	{attribute 'export' := '("archive":"True","communication":("cycle":"base","unsubscribe":["setpoint.LLV","setpoint.L1V","setpoint.LV","setpoint.HV","setpoint.H1V","setpoint.HHV"]),"journal":"True","name":("full":"Температура воздуха на входе осевого компрессора","short":"t на вх. Д"),"unit":("engineering":"°С","electrical":"°С"),"digit":"1","connection":("module":"UCP1-A1-AI7-5","type":"R","device_clamp":"UCP1","clamp":"XAI6:9A XAI6:9B XAI6:10B"),"subsystem":"Блок двигателя","group":["Блок двигателя"])'}
	Ta_inK : Taipar := (setpoint := (activation_flags := 0, hyst := GVL_LIB.Hyst_SP), cfg := (par_type := 4, lolim := -100, hilim := 200)); //Температура воздуха на входе осевого компрессора///Уставки//
END_VAR
(* global variable list aopar *)
{region INFO}
(*
 Назначение: Используется для хранения, инициализации и передачи на ВУ значений и состояния выходных аналоговых параметров
 Автор:      /Andrey/ 16.07.2025 17:15:05
 Версия ТЭ5: v00.00.01
 Проект:     KA107
*)
{endregion}
{attribute 'qualified_only'}
{attribute 'symbol' := 'readwrite'}
VAR_GLOBAL
	{attribute 'symbol' := 'none'}
	common : Taopar;
	{attribute 'export' := '("archive":"True","communication":("cycle":"fast"),"journal":"True","name":("full":"Управление положением дозатора газа"),"unit":("engineering":"%"),"connection":("module":"UCP1-A2-AO1-1","type":"I, акт.","device_clamp":"UCP1","clamp":"FVPP1:1 FVPP1:2"),"subsystem":"Блок двигателя","group":["Блок двигателя"])'}
	DG_set : Taopar := (cfg := (par_type := 1, lolim := 0, hilim := 100)); //Управление положением дозатора газа//
END_VAR
(* global variable list dipar *)
{region INFO}
(*
 Назначение: Используется для хранения, инициализации и передачи на ВУ значений и состояния входных дискретных параметров
 Автор:      /Andrey/ 16.07.2025 17:15:05
 Версия ТЭ5: v00.00.01
 Проект:     KA107
*)
{endregion}
{attribute 'qualified_only'}
{attribute 'symbol' := 'readwrite'}
VAR_GLOBAL
	{attribute 'symbol' := 'none'}
	common : Tdipar;

	{attribute 'symbol' := 'none'}
	AO_BA_ai : Tai_to_di;
	{attribute 'export' := '("archive":"True","communication":("cycle":"base"),"journal":"True","name":("full":"АО от блока автоматики ГПА"),"connection":("module":"UCP1-A2-DI1-01","type":"НО СК","device_clamp":"UCP1","clamp":"XDI1:1A XDI1:1B"),"subsystem":"Блок автоматики","group":["Блок автоматики"])'}
	AO_BA : Tdipar; //АО от блока автоматики ГПА//

	{attribute 'symbol' := 'none'}
	Fire_OD_ai : Tai_to_di;
	{attribute 'export' := '("archive":"True","communication":("cycle":"base"),"journal":"True","name":("full":"Пожар ОД"),"connection":("module":"UCP1-A2-DI1-02","type":"НО СК","device_clamp":"UCP1","clamp":"XDI1:2A XDI1:2B"),"subsystem":"Блок автоматики","group":["Блок автоматики"])'}
	Fire_OD : Tdipar; //Пожар ОД//

	{attribute 'symbol' := 'none'}
	Lm_MB_Pn_ai : Tai_to_di;
	{attribute 'export' := '("archive":"True","communication":("cycle":"base"),"journal":"True","name":("full":"Уровень масла в МБД+Н минимальный"),"connection":("module":"UCP1-A2-DI1-05","type":"НО СК","device_clamp":"UCP1","clamp":"XDI1:5A XDI1:5B"),"subsystem":"Маслосистема Д","group":["Маслосистема Д"])'}
	Lm_MB_Pn : Tdipar; //Уровень масла в МБД+Н минимальный//

	{attribute 'symbol' := 'none'}
	Lm_MBU_Pn_ai : Tai_to_di;
	{attribute 'export' := '("archive":"True","communication":("cycle":"base"),"journal":"True","name":("full":"Уровень масла в МБУпл. минимальный"),"connection":("module":"UCP1-A2-DI1-06","type":"НО СК","device_clamp":"UCP1","clamp":"XDI1:6A XDI1:6B"),"subsystem":"Маслосистема К","group":["Маслосистема К"])'}
	Lm_MBU_Pn : Tdipar; //Уровень масла в МБУпл. минимальный//

	{attribute 'symbol' := 'none'}
	Zagaz_OD_Pv_ai : Tai_to_di;
	{attribute 'export' := '("archive":"True","communication":("cycle":"base"),"journal":"True","name":("full":"Загазованность контейнеров выше нормы"),"connection":("module":"UCP1-A2-DI1-07","type":"НО СК","device_clamp":"UCP1","clamp":"XDI1:7A XDI1:7B"),"subsystem":"Блок автоматики","group":["Блок автоматики"])'}
	Zagaz_OD_Pv : Tdipar; //Загазованность контейнеров выше нормы//

	{attribute 'symbol' := 'none'}
	SurgeD_ai : Tai_to_di;
	{attribute 'export' := '("archive":"True","communication":("cycle":"base"),"journal":"True","name":("full":"Помпаж двигателя"),"connection":("module":"UCP1-A2-DI1-09","type":"НО СК","device_clamp":"UCP1","clamp":"XDI1:9A XDI1:9B"),"subsystem":"Блок двигателя","group":["Блок двигателя"])'}
	SurgeD : Tdipar; //Помпаж двигателя//

	{attribute 'symbol' := 'none'}
	Pm_TK_An_ai : Tai_to_di;
	{attribute 'export' := '("archive":"True","communication":("cycle":"base"),"journal":"True","name":("full":"Давление масла смазки ТК аварийная"),"connection":("module":"UCP1-A2-DI1-10","type":"НО СК","device_clamp":"UCP1","clamp":"XDI1:10A XDI1:10B"),"subsystem":"Блок двигателя","group":["Блок двигателя"])'}
	Pm_TK_An : Tdipar; //Давление масла смазки ТК аварийная//

	{attribute 'symbol' := 'none'}
	Pm_ST_An_ai : Tai_to_di;
	{attribute 'export' := '("archive":"True","communication":("cycle":"base"),"journal":"True","name":("full":"Давление масла смазки СТ аварийная"),"connection":("module":"UCP1-A2-DI1-11","type":"НО СК","device_clamp":"UCP1","clamp":"XDI1:11A XDI1:11B"),"subsystem":"Блок двигателя","group":["Блок двигателя"])'}
	Pm_ST_An : Tdipar; //Давление масла смазки СТ аварийная//

	{attribute 'symbol' := 'none'}
	Pm_N_An_ai : Tai_to_di;
	{attribute 'export' := '("archive":"True","communication":("cycle":"base"),"journal":"True","name":("full":"Давление масла смазки Н аварийная"),"connection":("module":"UCP1-A2-DI1-12","type":"НО СК","device_clamp":"UCP1","clamp":"XDI1:12A XDI1:12B"),"subsystem":"Блок компрессора","group":["Блок компрессора"])'}
	Pm_N_An : Tdipar; //Давление масла смазки Н аварийная//

	{attribute 'symbol' := 'none'}
	dPmg_An_ai : Tai_to_di;
	{attribute 'export' := '("archive":"True","communication":("cycle":"base"),"journal":"True","name":("full":"Аварийный перепад масло-газ"),"connection":("module":"UCP1-A2-DI1-13","type":"НО СК","device_clamp":"UCP1","clamp":"XDI1:13A XDI1:13B"),"subsystem":"Блок компрессора","group":["Блок компрессора"])'}
	dPmg_An : Tdipar; //Аварийный перепад масло-газ//

	{attribute 'symbol' := 'none'}
	Pm_SAR_An_ai : Tai_to_di;
	{attribute 'export' := '("archive":"True","communication":("cycle":"base"),"journal":"True","name":("full":"Давление масла САР < 1,5 МПа"),"connection":("module":"UCP1-A2-DI1-14","type":"НО СК","device_clamp":"UCP1","clamp":"XDI1:14A XDI1:14B"),"subsystem":"Блок двигателя","group":["Блок двигателя"])'}
	Pm_SAR_An : Tdipar; //Давление масла САР < 1,5 МПа//

	{attribute 'symbol' := 'none'}
	dP_F_Pv_ai : Tai_to_di;
	{attribute 'export' := '("archive":"True","communication":("cycle":"base"),"journal":"True","name":("full":"dP перед форсунками камеры сгорания >10кПа"),"connection":("module":"UCP1-A2-DI2-15","type":"НО СК","device_clamp":"UCP1","clamp":"FVD2:6 FVD2:5"),"subsystem":"Блок двигателя","group":["Блок двигателя"])'}
	dP_F_Pv : Tdipar; //dP перед форсунками камеры сгорания >10кПа//

	{attribute 'export' := '("archive":"True","communication":("cycle":"base"),"journal":"True","name":("full":"Вентилятор АВОМД+Н+У №1 включен"),"connection":("module":"UCP1-A2-DI3-3","type":"НО СК","device_clamp":"UCP1","clamp":"XDI2:3A XDI2:3B"),"subsystem":"АВОМ","group":["АВОМ"])'}
	Vn1_AVOM_ON : Tdipar; //Вентилятор АВОМД+Н+У №1 включен//
	{attribute 'export' := '("archive":"True","communication":("cycle":"base"),"journal":"True","name":("full":"Вентилятор АВОМД+Н+У №2 включен"),"connection":("module":"UCP1-A2-DI3-4","type":"НО СК","device_clamp":"UCP1","clamp":"XDI2:4A XDI2:4B"),"subsystem":"АВОМ","group":["АВОМ"])'}
	Vn2_AVOM_ON : Tdipar; //Вентилятор АВОМД+Н+У №2 включен//
	{attribute 'export' := '("archive":"True","communication":("cycle":"base"),"journal":"True","name":("full":"Вентилятор ВОУ включен"),"connection":("module":"UCP1-A2-DI3-5","type":"НО СК","device_clamp":"UCP1","clamp":"XDI2:5A XDI2:5B"),"subsystem":"Блок автоматики","group":["Блок автоматики"])'}
	VV_VOU_ON : Tdipar; //Вентилятор ВОУ включен//
	{attribute 'export' := '("archive":"True","communication":("cycle":"base"),"journal":"True","name":("full":"Вытяжной вентилятор нагнетателя ВВН включен"),"connection":("module":"UCP1-A2-DI3-6","type":"НО СК","device_clamp":"UCP1","clamp":"XDI2:6A XDI2:6B"),"subsystem":"Блок автоматики","group":["Блок автоматики"])'}
	VVN_ON : Tdipar; //Вытяжной вентилятор нагнетателя ВВН включен//
	{attribute 'export' := '("archive":"True","communication":("cycle":"base"),"journal":"True","name":("full":"ТРК: готовность"),"connection":("module":"UCP1-A2-DI3-9","type":"НО СК","device_clamp":"UCP1","clamp":"XDI2:9A XDI2:9B"),"subsystem":"Блок двигателя","group":["Блок двигателя"])'}
	TRKready : Tdipar; //ТРК: готовность//
	{attribute 'export' := '("archive":"True","communication":("cycle":"base"),"journal":"True","name":("full":"ТРК: авария"),"connection":("module":"UCP1-A2-DI3-10","type":"НЗ СК","device_clamp":"UCP1","clamp":"XDI2:10A XDI2:10B"),"subsystem":"Блок двигателя","group":["Блок двигателя"])'}
	TRKalr : Tdipar := (inv := TRUE); //ТРК: авария//
	{attribute 'export' := '("archive":"True","communication":("cycle":"base"),"journal":"True","name":("full":"Давление газа перед дозатором газа Предупредительное"),"connection":("module":"UCP1-A2-DI3-18","type":"НЗ СК","device_clamp":"UCP1","clamp":"XDI2:18A XDI2:18B"),"subsystem":"Блок двигателя","group":["Блок двигателя"])'}
	Ptg_inDG_Pn : Tdipar := (inv := TRUE); //Давление газа перед дозатором газа Предупредительное//
	{attribute 'export' := '("archive":"True","communication":("cycle":"base"),"journal":"True","name":("full":"Вентилятор АВОМД+Н+У №3 включен"),"connection":("module":"UCP1-A2-DI3-22","type":"НО СК","device_clamp":"UCP1","clamp":"XDI2:22A XDI2:22B"),"subsystem":"АВОМ","group":["АВОМ"])'}
	Vn3_AVOM_ON : Tdipar; //Вентилятор АВОМД+Н+У №3 включен//
	{attribute 'export' := '("archive":"True","communication":("cycle":"base"),"journal":"True","name":("full":"Вентилятор АВОМД+Н+У №4 включен"),"connection":("module":"UCP1-A2-DI3-23","type":"НО СК","device_clamp":"UCP1","clamp":"XDI2:23A XDI2:23B"),"subsystem":"АВОМ","group":["АВОМ"])'}
	Vn4_AVOM_ON : Tdipar; //Вентилятор АВОМД+Н+У №4 включен//
	{attribute 'export' := '("archive":"True","communication":("cycle":"base"),"journal":"True","name":("full":"Давление газа перед дозатором газа Аварийное"),"connection":("module":"UCP1-A2-DI3-24","type":"НО СК","device_clamp":"UCP1","clamp":"XDI2:24A XDI2:24B"),"subsystem":"Блок топливного газа","group":["Блок топливного газа"])'}
	Ptg_inDG_An : Tdipar; //Давление газа перед дозатором газа Аварийное//
	{attribute 'export' := '("archive":"True","communication":("cycle":"base"),"journal":"True","name":("full":"диаг. Предохранитель UCP1-XTFU1:1 питания модулей AO исправен"),"connection":("module":"UCP1-A2-DI4-17","type":"НО СК","device_clamp":"UCP1","clamp":"Внутр. сигнал"),"subsystem":"Блок автоматики","group":["Блок автоматики"])'}
	Fuse_AO_UCP1 : Tdipar; //диаг. Предохранитель UCP1-XTFU1:1 питания модулей AO исправен//
	{attribute 'export' := '("archive":"True","communication":("cycle":"base"),"journal":"True","name":("full":"диаг. Предохранитель UCP1-XTFU1:2 питания модулей DO исправен"),"connection":("module":"UCP1-A2-DI4-18","type":"НО СК","device_clamp":"UCP1","clamp":"Внутр. сигнал"),"subsystem":"Блок автоматики","group":["Блок автоматики"])'}
	Fuse_DO_UCP1 : Tdipar; //диаг. Предохранитель UCP1-XTFU1:2 питания модулей DO исправен//
	{attribute 'export' := '("archive":"True","communication":("cycle":"base"),"journal":"True","name":("full":"диаг. Предохранитель UCP1--XTFU6:1 питания датчиков температуры и влажности"),"connection":("module":"UCP1-A2-DI4-19","type":"НО СК","device_clamp":"UCP1","clamp":"Внутр. сигнал"),"subsystem":"Блок автоматики","group":["Блок автоматики"])'}
	Fuse_Air_UCP1 : Tdipar; //диаг. Предохранитель UCP1--XTFU6:1 питания датчиков температуры и влажности//
	{attribute 'symbol' := 'none'}
	AO_PRU_1_ai : Tai_to_di;
	{attribute 'export' := '("archive":"True","communication":("cycle":"base"),"journal":"True","name":("full":"Кнопка АО на ПРУ сигнал 1 (НР)"),"connection":("module":"UE1-A1-DI1-01","type":"НО СК","device_clamp":"UE1","clamp":"XTH1:4 XTH1:3"),"subsystem":"Блок автоматики","group":["Блок автоматики"])'}
	AO_PRU_1 : Tdipar; //Кнопка АО на ПРУ сигнал 1 (НР)//

	{attribute 'symbol' := 'none'}
	Kr1_off_ai : Tai_to_di;
	{attribute 'export' := '("archive":"True","communication":("cycle":"base"),"journal":"True","name":("full":"Кран 1 закрыт"),"connection":("module":"UE1-A1-DI1-02","type":"НО СК","device_clamp":"UE1","clamp":"XDI1:2A XDI1:2B"),"subsystem":"Газовая обвязка","group":["Газовая обвязка"])'}
	Kr1_off : Tdipar; //Кран 1 закрыт//

	{attribute 'symbol' := 'none'}
	Kr2_off_ai : Tai_to_di;
	{attribute 'export' := '("archive":"True","communication":("cycle":"base"),"journal":"True","name":("full":"Кран 2 закрыт"),"connection":("module":"UE1-A1-DI1-03","type":"НО СК","device_clamp":"UE1","clamp":"XDI1:3A XDI1:3B"),"subsystem":"Газовая обвязка","group":["Газовая обвязка"])'}
	Kr2_off : Tdipar; //Кран 2 закрыт//

	{attribute 'symbol' := 'none'}
	Kr4_off_ai : Tai_to_di;
	{attribute 'export' := '("archive":"True","communication":("cycle":"base"),"journal":"True","name":("full":"Кран 4 закрыт"),"connection":("module":"UE1-A1-DI1-04","type":"НО СК","device_clamp":"UE1","clamp":"XDI1:4A XDI1:4B"),"subsystem":"Газовая обвязка","group":["Газовая обвязка"])'}
	Kr4_off : Tdipar; //Кран 4 закрыт//

	{attribute 'symbol' := 'none'}
	Kr5_off_ai : Tai_to_di;
	{attribute 'export' := '("archive":"True","communication":("cycle":"base"),"journal":"True","name":("full":"Кран 5 закрыт"),"connection":("module":"UE1-A1-DI1-05","type":"НО СК","device_clamp":"UE1","clamp":"XDI1:5A XDI1:5B"),"subsystem":"Газовая обвязка","group":["Газовая обвязка"])'}
	Kr5_off : Tdipar; //Кран 5 закрыт//

	{attribute 'symbol' := 'none'}
	Kr6_off_ai : Tai_to_di;
	{attribute 'export' := '("archive":"True","communication":("cycle":"base"),"journal":"True","name":("full":"Кран 6 закрыт"),"connection":("module":"UE1-A1-DI1-06","type":"НО СК","device_clamp":"UE1","clamp":"XDI1:6A XDI1:6B"),"subsystem":"Газовая обвязка","group":["Газовая обвязка"])'}
	Kr6_off : Tdipar; //Кран 6 закрыт//

	{attribute 'symbol' := 'none'}
	Kr12_off_ai : Tai_to_di;
	{attribute 'export' := '("archive":"True","communication":("cycle":"base"),"journal":"True","name":("full":"Кран 12 закрыт (т.г.)"),"connection":("module":"UE1-A1-DI1-07","type":"НО СК","device_clamp":"UE1","clamp":"XDI1:7A XDI1:7B"),"subsystem":"Газовая обвязка","group":["Газовая обвязка"])'}
	Kr12_off : Tdipar; //Кран 12 закрыт (т.г.)//

	{attribute 'symbol' := 'none'}
	Kr9_off_ai : Tai_to_di;
	{attribute 'export' := '("archive":"True","communication":("cycle":"base"),"journal":"True","name":("full":"Кран 9 закрыт (т.газ. свеча.)"),"connection":("module":"UE1-A1-DI1-08","type":"НО СК","device_clamp":"UE1","clamp":"XDI1:8A XDI1:8B"),"subsystem":"Газовая обвязка","group":["Газовая обвязка"])'}
	Kr9_off : Tdipar; //Кран 9 закрыт (т.газ. свеча.)//

	{attribute 'symbol' := 'none'}
	Kr11_off_ai : Tai_to_di;
	{attribute 'export' := '("archive":"True","communication":("cycle":"base"),"journal":"True","name":("full":"Кран 11 закрыт (п.г.)"),"connection":("module":"UE1-A1-DI1-09","type":"НО СК","device_clamp":"UE1","clamp":"XDI1:9A XDI1:9B"),"subsystem":"Газовая обвязка","group":["Газовая обвязка"])'}
	Kr11_off : Tdipar; //Кран 11 закрыт (п.г.)//

	{attribute 'symbol' := 'none'}
	Kr10_off_ai : Tai_to_di;
	{attribute 'export' := '("archive":"True","communication":("cycle":"base"),"journal":"True","name":("full":"Кран 10 закрыт (п.газ. свеча.)"),"connection":("module":"UE1-A1-DI1-10","type":"НО СК","device_clamp":"UE1","clamp":"XDI1:10A XDI1:10B"),"subsystem":"Газовая обвязка","group":["Газовая обвязка"])'}
	Kr10_off : Tdipar; //Кран 10 закрыт (п.газ. свеча.)//

	{attribute 'symbol' := 'none'}
	KPV1_off_ai : Tai_to_di;
	{attribute 'export' := '("archive":"True","communication":("cycle":"base"),"journal":"True","name":("full":"КПВ-1 закрыт"),"connection":("module":"UE1-A1-DI1-11","type":"НО СК","device_clamp":"UE1","clamp":"XDI1:11A XDI1:11B"),"subsystem":"Блок двигателя","group":["Блок двигателя"])'}
	KPV1_off : Tdipar; //КПВ-1 закрыт//

	{attribute 'symbol' := 'none'}
	KPV2_off_ai : Tai_to_di;
	{attribute 'export' := '("archive":"True","communication":("cycle":"base"),"journal":"True","name":("full":"КПВ-2 закрыт"),"connection":("module":"UE1-A1-DI1-12","type":"НО СК","device_clamp":"UE1","clamp":"XDI1:12A XDI1:12B"),"subsystem":"Блок двигателя","group":["Блок двигателя"])'}
	KPV2_off : Tdipar; //КПВ-2 закрыт//

	{attribute 'symbol' := 'none'}
	KPV3_off_ai : Tai_to_di;
	{attribute 'export' := '("archive":"True","communication":("cycle":"base"),"journal":"True","name":("full":"КПВ-3 закрыт"),"connection":("module":"UE1-A1-DI1-13","type":"НО СК","device_clamp":"UE1","clamp":"XDI1:13A XDI1:13B"),"subsystem":"Блок двигателя","group":["Блок двигателя"])'}
	KPV3_off : Tdipar; //КПВ-3 закрыт//

	{attribute 'symbol' := 'none'}
	KPV4_off_ai : Tai_to_di;
	{attribute 'export' := '("archive":"True","communication":("cycle":"base"),"journal":"True","name":("full":"КПВ-4 закрыт"),"connection":("module":"UE1-A1-DI1-14","type":"НО СК","device_clamp":"UE1","clamp":"XDI1:14A XDI1:14B"),"subsystem":"Блок двигателя","group":["Блок двигателя"])'}
	KPV4_off : Tdipar; //КПВ-4 закрыт//

	{attribute 'symbol' := 'none'}
	KPV5_off_ai : Tai_to_di;
	{attribute 'export' := '("archive":"True","communication":("cycle":"base"),"journal":"True","name":("full":"КПВ-5 закрыт"),"connection":("module":"UE1-A1-DI1-15","type":"НО СК","device_clamp":"UE1","clamp":"XDI1:15A XDI1:15B"),"subsystem":"Блок двигателя","group":["Блок двигателя"])'}
	KPV5_off : Tdipar; //КПВ-5 закрыт//

	{attribute 'symbol' := 'none'}
	SK_off_ai : Tai_to_di;
	{attribute 'export' := '("archive":"True","communication":("cycle":"fast"),"journal":"True","name":("full":"СК закрыт"),"connection":("module":"UE1-A1-DI1-16","type":"НО СК","device_clamp":"UE1","clamp":"XDI1:16A XDI1:16B"),"subsystem":"Блок топливного газа","group":["Блок топливного газа"])'}
	SK_off : Tdipar; //СК закрыт//

	{attribute 'symbol' := 'none'}
	AO_PRU_2_ai : Tai_to_di;
	{attribute 'export' := '("archive":"True","communication":("cycle":"base"),"journal":"True","name":("full":"Кнопка АО на ПРУ сигнал 2 (НЗ)"),"connection":("module":"UE1-A1-DI2-01","type":"НЗ СК","device_clamp":"UE1","clamp":"XTH1:13 XTH1:14"),"subsystem":"Блок автоматики","group":["Блок автоматики"])'}
	AO_PRU_2 : Tdipar := (inv := TRUE); //Кнопка АО на ПРУ сигнал 2 (НЗ)//

	{attribute 'symbol' := 'none'}
	Kr1_ON_ai : Tai_to_di;
	{attribute 'export' := '("archive":"True","communication":("cycle":"base"),"journal":"True","name":("full":"Кран 1 открыт"),"connection":("module":"UE1-A1-DI2-02","type":"НО СК","device_clamp":"UE1","clamp":"XDI1:18A XDI1:18B"),"subsystem":"Газовая обвязка","group":["Газовая обвязка"])'}
	Kr1_ON : Tdipar; //Кран 1 открыт//

	{attribute 'symbol' := 'none'}
	Kr2_ON_ai : Tai_to_di;
	{attribute 'export' := '("archive":"True","communication":("cycle":"base"),"journal":"True","name":("full":"Кран 2 открыт"),"connection":("module":"UE1-A1-DI2-03","type":"НО СК","device_clamp":"UE1","clamp":"XDI1:19A XDI1:19B"),"subsystem":"Газовая обвязка","group":["Газовая обвязка"])'}
	Kr2_ON : Tdipar; //Кран 2 открыт//

	{attribute 'symbol' := 'none'}
	Kr4_ON_ai : Tai_to_di;
	{attribute 'export' := '("archive":"True","communication":("cycle":"base"),"journal":"True","name":("full":"Кран 4 открыт"),"connection":("module":"UE1-A1-DI2-04","type":"НО СК","device_clamp":"UE1","clamp":"XDI1:20A XDI1:20B"),"subsystem":"Газовая обвязка","group":["Газовая обвязка"])'}
	Kr4_ON : Tdipar; //Кран 4 открыт//

	{attribute 'symbol' := 'none'}
	Kr5_ON_ai : Tai_to_di;
	{attribute 'export' := '("archive":"True","communication":("cycle":"base"),"journal":"True","name":("full":"Кран 5 открыт"),"connection":("module":"UE1-A1-DI2-05","type":"НО СК","device_clamp":"UE1","clamp":"XDI1:21A XDI1:21B"),"subsystem":"Газовая обвязка","group":["Газовая обвязка"])'}
	Kr5_ON : Tdipar; //Кран 5 открыт//

	{attribute 'symbol' := 'none'}
	Kr6_ON_ai : Tai_to_di;
	{attribute 'export' := '("archive":"True","communication":("cycle":"base"),"journal":"True","name":("full":"Кран 6 открыт"),"connection":("module":"UE1-A1-DI2-06","type":"НО СК","device_clamp":"UE1","clamp":"XDI1:22A XDI1:22B"),"subsystem":"Газовая обвязка","group":["Газовая обвязка"])'}
	Kr6_ON : Tdipar; //Кран 6 открыт//

	{attribute 'symbol' := 'none'}
	Kr12_ON_ai : Tai_to_di;
	{attribute 'export' := '("archive":"True","communication":("cycle":"base"),"journal":"True","name":("full":"Кран 12 открыт (т.г.)"),"connection":("module":"UE1-A1-DI2-07","type":"НО СК","device_clamp":"UE1","clamp":"XDI1:23A XDI1:23B"),"subsystem":"Газовая обвязка","group":["Газовая обвязка"])'}
	Kr12_ON : Tdipar; //Кран 12 открыт (т.г.)//

	{attribute 'symbol' := 'none'}
	Kr9_ON_ai : Tai_to_di;
	{attribute 'export' := '("archive":"True","communication":("cycle":"base"),"journal":"True","name":("full":"Кран 9 открыт (т.газ. свеча.)"),"connection":("module":"UE1-A1-DI2-08","type":"НО СК","device_clamp":"UE1","clamp":"XDI1:24A XDI1:24B"),"subsystem":"Газовая обвязка","group":["Газовая обвязка"])'}
	Kr9_ON : Tdipar; //Кран 9 открыт (т.газ. свеча.)//

	{attribute 'symbol' := 'none'}
	Kr11_ON_ai : Tai_to_di;
	{attribute 'export' := '("archive":"True","communication":("cycle":"base"),"journal":"True","name":("full":"Кран 11 открыт (п.г.)"),"connection":("module":"UE1-A1-DI2-09","type":"НО СК","device_clamp":"UE1","clamp":"XDI1:25A XDI1:25B"),"subsystem":"Газовая обвязка","group":["Газовая обвязка"])'}
	Kr11_ON : Tdipar; //Кран 11 открыт (п.г.)//

	{attribute 'symbol' := 'none'}
	Kr10_ON_ai : Tai_to_di;
	{attribute 'export' := '("archive":"True","communication":("cycle":"base"),"journal":"True","name":("full":"Кран 10 открыт (п.газ. свеча.)"),"connection":("module":"UE1-A1-DI2-10","type":"НО СК","device_clamp":"UE1","clamp":"XDI1:26A XDI1:26B"),"subsystem":"Газовая обвязка","group":["Газовая обвязка"])'}
	Kr10_ON : Tdipar; //Кран 10 открыт (п.газ. свеча.)//

	{attribute 'symbol' := 'none'}
	KPV1_ON_ai : Tai_to_di;
	{attribute 'export' := '("archive":"True","communication":("cycle":"base"),"journal":"True","name":("full":"КПВ-1 открыт"),"connection":("module":"UE1-A1-DI2-11","type":"НО СК","device_clamp":"UE1","clamp":"XDI1:27A XDI1:27B"),"subsystem":"Блок двигателя","group":["Блок двигателя"])'}
	KPV1_ON : Tdipar; //КПВ-1 открыт//

	{attribute 'symbol' := 'none'}
	KPV2_ON_ai : Tai_to_di;
	{attribute 'export' := '("archive":"True","communication":("cycle":"base"),"journal":"True","name":("full":"КПВ-2 открыт"),"connection":("module":"UE1-A1-DI2-12","type":"НО СК","device_clamp":"UE1","clamp":"XDI1:28A XDI1:28B"),"subsystem":"Блок двигателя","group":["Блок двигателя"])'}
	KPV2_ON : Tdipar; //КПВ-2 открыт//

	{attribute 'symbol' := 'none'}
	KPV3_ON_ai : Tai_to_di;
	{attribute 'export' := '("archive":"True","communication":("cycle":"base"),"journal":"True","name":("full":"КПВ-3 открыт"),"connection":("module":"UE1-A1-DI2-13","type":"НО СК","device_clamp":"UE1","clamp":"XDI1:29A XDI1:29B"),"subsystem":"Блок двигателя","group":["Блок двигателя"])'}
	KPV3_ON : Tdipar; //КПВ-3 открыт//

	{attribute 'symbol' := 'none'}
	KPV4_ON_ai : Tai_to_di;
	{attribute 'export' := '("archive":"True","communication":("cycle":"base"),"journal":"True","name":("full":"КПВ-4 открыт"),"connection":("module":"UE1-A1-DI2-14","type":"НО СК","device_clamp":"UE1","clamp":"XDI1:30A XDI1:30B"),"subsystem":"Блок двигателя","group":["Блок двигателя"])'}
	KPV4_ON : Tdipar; //КПВ-4 открыт//

	{attribute 'symbol' := 'none'}
	KPV5_ON_ai : Tai_to_di;
	{attribute 'export' := '("archive":"True","communication":("cycle":"base"),"journal":"True","name":("full":"КПВ-5 открыт"),"connection":("module":"UE1-A1-DI2-15","type":"НО СК","device_clamp":"UE1","clamp":"XDI1:31A XDI1:31B"),"subsystem":"Блок двигателя","group":["Блок двигателя"])'}
	KPV5_ON : Tdipar; //КПВ-5 открыт//

	{attribute 'symbol' := 'none'}
	SK_ON_ai : Tai_to_di;
	{attribute 'export' := '("archive":"True","communication":("cycle":"fast"),"journal":"True","name":("full":"СК открыт"),"connection":("module":"UE1-A1-DI2-16","type":"НО СК","device_clamp":"UE1","clamp":"XDI1:32A XDI1:32B"),"subsystem":"Блок топливного газа","group":["Блок топливного газа"])'}
	SK_ON : Tdipar; //СК открыт//

	{attribute 'symbol' := 'none'}
	PNS_ON_ai : Tai_to_di;
	{attribute 'export' := '("archive":"True","communication":("cycle":"base"),"journal":"True","name":("full":"Пусковой насос смазки включен"),"connection":("module":"UE1-A1-DI3-01","type":"НО СК","device_clamp":"UE1","clamp":"XDI2:1A XDI2:1B"),"subsystem":"Маслосистема Д","group":["Маслосистема Д"])'}
	PNS_ON : Tdipar; //Пусковой насос смазки включен//

	{attribute 'symbol' := 'none'}
	PNU_ON_ai : Tai_to_di;
	{attribute 'export' := '("archive":"True","communication":("cycle":"base"),"journal":"True","name":("full":"Пусковой насос уплотнения включен"),"connection":("module":"UE1-A1-DI3-02","type":"НО СК","device_clamp":"UE1","clamp":"XDI2:2A XDI2:2B"),"subsystem":"Маслосистема К","group":["Маслосистема К"])'}
	PNU_ON : Tdipar; //Пусковой насос уплотнения включен//

	{attribute 'export' := '("archive":"True","communication":("cycle":"base"),"journal":"True","name":("full":"Повышенная вибрация двигателя"),"connection":("module":"UE1-A1-DI4-9","type":"НО СК","device_clamp":"UE1","clamp":"XDI3:9A XDI3:9B"),"subsystem":"Блок двигателя","group":["Блок двигателя"])'}
	Vs_D_Pv : Tdipar; //Повышенная вибрация двигателя//
	{attribute 'export' := '("archive":"True","communication":("cycle":"base"),"journal":"True","name":("full":"Опасная вибрация двигателя"),"connection":("module":"UE1-A1-DI4-10","type":"НО СК","device_clamp":"UE1","clamp":"XDI3:10A XDI3:10B"),"subsystem":"Блок двигателя","group":["Блок двигателя"])'}
	Vs_D_Av : Tdipar; //Опасная вибрация двигателя//
	{attribute 'export' := '("archive":"True","communication":("cycle":"base"),"journal":"True","name":("full":"Осевой сдвиг ротора Н Аварийный"),"connection":("module":"UE1-A1-DI4-18","type":"НО СК","device_clamp":"UE1","clamp":"XDI3:18A XDI3:18B"),"subsystem":"Блок компрессора","group":["Блок компрессора"])'}
	Zs_Nl : Tdipar; //Осевой сдвиг ротора Н Аварийный//
	{attribute 'export' := '("archive":"True","communication":("cycle":"base"),"journal":"True","name":("full":"Давление газа после крана 1"),"connection":("module":"UE1-A1-DI4-20","type":"НО СК","device_clamp":"UE1","clamp":"XDI3:20A XDI3:20B"),"subsystem":"Газовая обвязка","group":["Газовая обвязка"])'}
	Pg_outKR1 : Tdipar; //Давление газа после крана 1//
	{attribute 'export' := '("archive":"True","communication":("cycle":"base"),"journal":"True","name":("full":"Давление масла смазки Н предупредительная"),"connection":("module":"UE1-A1-DI4-23","type":"НО СК","device_clamp":"UE1","clamp":"XDI3:23A XDI3:23B"),"subsystem":"Маслосистема К","group":["Маслосистема К"])'}
	Pm_N_Pn : Tdipar; //Давление масла смазки Н предупредительная//
	{attribute 'export' := '("archive":"True","communication":("cycle":"base"),"journal":"True","name":("full":"Разрежение в ВОУ"),"connection":("module":"UE1-A1-DI4-24","type":"НО СК","device_clamp":"UE1","clamp":"XDI3:24A XDI3:24B"),"subsystem":"Блок двигателя","group":["Блок двигателя"])'}
	Exh_VOU : Tdipar; //Разрежение в ВОУ//
	{attribute 'export' := '("archive":"True","communication":("cycle":"base"),"journal":"True","name":("full":"Давление газа до крана 13 (воздушного стартера)"),"connection":("module":"UE1-A1-DI4-25","type":"НО СК","device_clamp":"UE1","clamp":"XDI3:25A XDI3:25B"),"subsystem":"Газовая обвязка","group":["Газовая обвязка"])'}
	Pg_InKR13 : Tdipar; //Давление газа до крана 13 (воздушного стартера)//
	{attribute 'export' := '("archive":"True","communication":("cycle":"base"),"journal":"True","name":("full":"Давление масла смазки воздушного стартера высокий уровень"),"connection":("module":"UE1-A1-DI4-26","type":"НО СК","device_clamp":"UE1","clamp":"XDI3:26A XDI3:26B"),"subsystem":"Маслосистема Д","group":["Маслосистема Д"])'}
	Pm_Starter_Av : Tdipar; //Давление масла смазки воздушного стартера высокий уровень//
	{attribute 'export' := '("archive":"True","communication":("cycle":"base"),"journal":"True","name":("full":"Давление масла смазки воздушного стартера низкий уровень"),"connection":("module":"UE1-A1-DI4-27","type":"НО СК","device_clamp":"UE1","clamp":"XDI3:27A XDI3:27B"),"subsystem":"Маслосистема Д","group":["Маслосистема Д"])'}
	Pm_Starter_An : Tdipar; //Давление масла смазки воздушного стартера низкий уровень//
	{attribute 'export' := '("archive":"True","communication":("cycle":"base"),"journal":"True","name":("full":"Кнопка ЭАО на ПРУ нажата сигнал 1 (НР)"),"connection":("module":"UE1-A1-DI4-29","type":"НО СК","device_clamp":"UE1","clamp":"Внутр. сигнал"),"subsystem":"Блок автоматики","group":["Блок автоматики"])'}
	EAO_PRU_1 : Tdipar; //Кнопка ЭАО на ПРУ нажата сигнал 1 (НР)//
	{attribute 'export' := '("archive":"True","communication":("cycle":"base"),"journal":"True","name":("full":"Кнопка ЭАО на ПРУ нажата сигнал 2 (НЗ)"),"connection":("module":"UE1-A1-DI4-30","type":"НЗ СК","device_clamp":"UE1","clamp":"Внутр. сигнал"),"subsystem":"Блок автоматики","group":["Блок автоматики"])'}
	EAO_PRU_2 : Tdipar := (inv := TRUE); //Кнопка ЭАО на ПРУ нажата сигнал 2 (НЗ)//
	{attribute 'export' := '("archive":"True","communication":("cycle":"base"),"journal":"True","name":("full":"Кнопка ЭАО на ПРУ нажата сигнал 3 (НЗ)"),"connection":("module":"UE1-A1-DI4-31","type":"НЗ СК","device_clamp":"UE1","clamp":"Внутр. сигнал"),"subsystem":"Блок автоматики","group":["Блок автоматики"])'}
	EAO_PRU_3 : Tdipar := (inv := TRUE); //Кнопка ЭАО на ПРУ нажата сигнал 3 (НЗ)//
	{attribute 'export' := '("archive":"True","communication":("cycle":"base"),"journal":"True","name":("full":"БЭАО сработал"),"connection":("module":"UE1-A1-DI4-32","type":"НО СК","device_clamp":"UE1","clamp":"Внутр. сигнал"),"subsystem":"Блок автоматики","group":["Блок автоматики"])'}
	BEAO : Tdipar; //БЭАО сработал//
	{attribute 'export' := '("archive":"True","communication":("cycle":"base"),"journal":"True","name":("full":"Заслонка ВC (кран 13) открыта"),"connection":("module":"UE1-A1-DI5-1","type":"U","device_clamp":"UE1","clamp":"DA1:A2"),"subsystem":"Газовая обвязка","group":["Газовая обвязка"])'}
	Kr13_ON : Tdipar; //Заслонка ВC (кран 13) открыта//
	{attribute 'export' := '("archive":"True","communication":("cycle":"base"),"journal":"True","name":("full":"БЗА. Авария"),"connection":("module":"UE1-A1-DI5-2","type":"НО СК","device_clamp":"UE1","clamp":"Внутр. сигнал"),"subsystem":"Блок автоматики","group":["Блок автоматики"])'}
	BZA_alr : Tdipar; //БЗА. Авария//
	{attribute 'export' := '("archive":"True","communication":("cycle":"base"),"journal":"True","name":("full":"БЗА. Готовность 1"),"connection":("module":"UE1-A1-DI5-3","type":"НО СК","device_clamp":"UE1","clamp":"Внутр. сигнал"),"subsystem":"Блок автоматики","group":["Блок автоматики"])'}
	BZA_ready_1 : Tdipar; //БЗА. Готовность 1//
	{attribute 'export' := '("archive":"True","communication":("cycle":"base"),"journal":"True","name":("full":"БЗА. Готовность 2"),"connection":("module":"UE1-A1-DI5-4","type":"НО СК","device_clamp":"UE1","clamp":"Внутр. сигнал"),"subsystem":"Блок автоматики","group":["Блок автоматики"])'}
	BZA_ready_2 : Tdipar; //БЗА. Готовность 2//
	{attribute 'export' := '("archive":"True","communication":("cycle":"base"),"journal":"True","name":("full":"Контроль питания СС"),"connection":("module":"UE1-A1-DI5-25","type":"НО СК","device_clamp":"UE1","clamp":"Внутр. сигнал"),"subsystem":"Блок автоматики","group":["Блок автоматики"])'}
	U_CC_cntrl : Tdipar; //Контроль питания СС//
	{attribute 'export' := '("archive":"True","communication":("cycle":"base"),"journal":"True","name":("full":"Стружка в масле на выходе Д"),"connection":("module":"UE1-A1-DI5-26","type":"НО СК","device_clamp":"UE1","clamp":"XDI4:26A XDI4:26B"),"subsystem":"Маслосистема Д","group":["Маслосистема Д"])'}
	Chip_outD : Tdipar; //Стружка в масле на выходе Д//
	{attribute 'export' := '("archive":"True","communication":("cycle":"base"),"journal":"True","name":("full":"Сигнализатор обледенения"),"connection":("module":"UE1-A1-DI5-27","type":"НО СК","device_clamp":"UE1","clamp":"XDI4:27A XDI4:27B"),"subsystem":"Блок автоматики","group":["Блок автоматики"])'}
	Ace_alr : Tdipar; //Сигнализатор обледенения//
	{attribute 'export' := '("archive":"True","communication":("cycle":"base"),"journal":"True","name":("full":"диаг. Кран 1 закрыть"),"connection":("module":"UE1-A1-DI6-1","type":"НО СК","device_clamp":"UE1","clamp":"Внутр. сигнал"),"subsystem":"Газовая обвязка","group":["Газовая обвязка"])'}
	kcdo_Kr1_off : Tdipar; //диаг. Кран 1 закрыть//
	{attribute 'export' := '("archive":"True","communication":("cycle":"base"),"journal":"True","name":("full":"диаг. Кран 1 смазка"),"connection":("module":"UE1-A1-DI6-2","type":"НО СК","device_clamp":"UE1","clamp":"Внутр. сигнал"),"subsystem":"Газовая обвязка","group":["Газовая обвязка"])'}
	kcdo_Kr1m_ON : Tdipar; //диаг. Кран 1 смазка//
	{attribute 'export' := '("archive":"True","communication":("cycle":"base"),"journal":"True","name":("full":"диаг. Кран 2 закрыть"),"connection":("module":"UE1-A1-DI6-3","type":"НО СК","device_clamp":"UE1","clamp":"Внутр. сигнал"),"subsystem":"Газовая обвязка","group":["Газовая обвязка"])'}
	kcdo_Kr2_off : Tdipar; //диаг. Кран 2 закрыть//
	{attribute 'export' := '("archive":"True","communication":("cycle":"base"),"journal":"True","name":("full":"диаг. Кран 2 смазка"),"connection":("module":"UE1-A1-DI6-4","type":"НО СК","device_clamp":"UE1","clamp":"Внутр. сигнал"),"subsystem":"Газовая обвязка","group":["Газовая обвязка"])'}
	kcdo_Kr2m_ON : Tdipar; //диаг. Кран 2 смазка//
	{attribute 'export' := '("archive":"True","communication":("cycle":"base"),"journal":"True","name":("full":"диаг. Кран 4 закрыть"),"connection":("module":"UE1-A1-DI6-5","type":"НО СК","device_clamp":"UE1","clamp":"Внутр. сигнал"),"subsystem":"Газовая обвязка","group":["Газовая обвязка"])'}
	kcdo_Kr4_off : Tdipar; //диаг. Кран 4 закрыть//
	{attribute 'export' := '("archive":"True","communication":("cycle":"base"),"journal":"True","name":("full":"диаг. Кран 4 смазка"),"connection":("module":"UE1-A1-DI6-6","type":"НО СК","device_clamp":"UE1","clamp":"Внутр. сигнал"),"subsystem":"Газовая обвязка","group":["Газовая обвязка"])'}
	kcdo_Kr4m_ON : Tdipar; //диаг. Кран 4 смазка//
	{attribute 'export' := '("archive":"True","communication":("cycle":"base"),"journal":"True","name":("full":"диаг. Кран 5 открыть"),"connection":("module":"UE1-A1-DI6-7","type":"НО СК","device_clamp":"UE1","clamp":"Внутр. сигнал"),"subsystem":"Газовая обвязка","group":["Газовая обвязка"])'}
	kcdo_Kr5_ON : Tdipar; //диаг. Кран 5 открыть//
	{attribute 'export' := '("archive":"True","communication":("cycle":"base"),"journal":"True","name":("full":"диаг. Кран 5 смазка"),"connection":("module":"UE1-A1-DI6-8","type":"НО СК","device_clamp":"UE1","clamp":"Внутр. сигнал"),"subsystem":"Газовая обвязка","group":["Газовая обвязка"])'}
	kcdo_Kr5m_ON : Tdipar; //диаг. Кран 5 смазка//
	{attribute 'export' := '("archive":"True","communication":("cycle":"base"),"journal":"True","name":("full":"диаг. Кран 6 закрыть"),"connection":("module":"UE1-A1-DI6-9","type":"НО СК","device_clamp":"UE1","clamp":"Внутр. сигнал"),"subsystem":"Газовая обвязка","group":["Газовая обвязка"])'}
	kcdo_Kr6_off : Tdipar; //диаг. Кран 6 закрыть//
	{attribute 'export' := '("archive":"True","communication":("cycle":"base"),"journal":"True","name":("full":"диаг. Кран 6 смазка"),"connection":("module":"UE1-A1-DI6-10","type":"НО СК","device_clamp":"UE1","clamp":"Внутр. сигнал"),"subsystem":"Газовая обвязка","group":["Газовая обвязка"])'}
	kcdo_Kr6m_ON : Tdipar; //диаг. Кран 6 смазка//
	{attribute 'export' := '("archive":"True","communication":("cycle":"base"),"journal":"True","name":("full":"диаг. Кран 12 закрыть (т.г.)"),"connection":("module":"UE1-A1-DI6-11","type":"НО СК","device_clamp":"UE1","clamp":"Внутр. сигнал"),"subsystem":"Газовая обвязка","group":["Газовая обвязка"])'}
	kcdo_KR12_off : Tdipar; //диаг. Кран 12 закрыть (т.г.)//
	{attribute 'export' := '("archive":"True","communication":("cycle":"base"),"journal":"True","name":("full":"диаг. Кран 12 смазка"),"connection":("module":"UE1-A1-DI6-12","type":"НО СК","device_clamp":"UE1","clamp":"Внутр. сигнал"),"subsystem":"Газовая обвязка","group":["Газовая обвязка"])'}
	kcdo_KR12m_ON : Tdipar; //диаг. Кран 12 смазка//
	{attribute 'export' := '("archive":"True","communication":("cycle":"base"),"journal":"True","name":("full":"диаг. Кран 9 смазка"),"connection":("module":"UE1-A1-DI6-14","type":"НО СК","device_clamp":"UE1","clamp":"Внутр. сигнал"),"subsystem":"Газовая обвязка","group":["Газовая обвязка"])'}
	kcdo_KR9m_ON : Tdipar; //диаг. Кран 9 смазка//
	{attribute 'export' := '("archive":"True","communication":("cycle":"base"),"journal":"True","name":("full":"диаг. Кран 11 открыть (п.г.)"),"connection":("module":"UE1-A1-DI6-15","type":"НО СК","device_clamp":"UE1","clamp":"Внутр. сигнал"),"subsystem":"Газовая обвязка","group":["Газовая обвязка"])'}
	kcdo_Kr11_ON : Tdipar; //диаг. Кран 11 открыть (п.г.)//
	{attribute 'export' := '("archive":"True","communication":("cycle":"base"),"journal":"True","name":("full":"диаг. Кран 11 смазка"),"connection":("module":"UE1-A1-DI6-16","type":"НО СК","device_clamp":"UE1","clamp":"Внутр. сигнал"),"subsystem":"Газовая обвязка","group":["Газовая обвязка"])'}
	kcdo_Kr11m_ON : Tdipar; //диаг. Кран 11 смазка//
	{attribute 'export' := '("archive":"True","communication":("cycle":"base"),"journal":"True","name":("full":"диаг. Кран 10 смазка"),"connection":("module":"UE1-A1-DI6-18","type":"НО СК","device_clamp":"UE1","clamp":"Внутр. сигнал"),"subsystem":"Газовая обвязка","group":["Газовая обвязка"])'}
	kcdo_Kr10m_ON : Tdipar; //диаг. Кран 10 смазка//
	{attribute 'export' := '("archive":"True","communication":("cycle":"base"),"journal":"True","name":("full":"диаг. Включение КПВ 1,5"),"connection":("module":"UE1-A1-DI6-19","type":"НО СК","device_clamp":"UE1","clamp":"Внутр. сигнал"),"subsystem":"Блок двигателя","group":["Блок двигателя"])'}
	kcdo_KPV15_ON : Tdipar; //диаг. Включение КПВ 1,5//
	{attribute 'export' := '("archive":"True","communication":("cycle":"base"),"journal":"True","name":("full":"диаг. Включение КПВ 2,3"),"connection":("module":"UE1-A1-DI6-20","type":"НО СК","device_clamp":"UE1","clamp":"Внутр. сигнал"),"subsystem":"Блок двигателя","group":["Блок двигателя"])'}
	kcdo_KPV23_off : Tdipar; //диаг. Включение КПВ 2,3//
	{attribute 'export' := '("archive":"True","communication":("cycle":"base"),"journal":"True","name":("full":"диаг. Включение КПВ 4"),"connection":("module":"UE1-A1-DI6-21","type":"НО СК","device_clamp":"UE1","clamp":"Внутр. сигнал"),"subsystem":"Блок двигателя","group":["Блок двигателя"])'}
	kcdo_KPV4_off : Tdipar; //диаг. Включение КПВ 4//
	{attribute 'export' := '("archive":"True","communication":("cycle":"base"),"journal":"True","name":("full":"диаг. Стопорный клапан открыть"),"connection":("module":"UE1-A1-DI6-22","type":"НО СК","device_clamp":"UE1","clamp":"Внутр. сигнал"),"subsystem":"Блок двигателя","group":["Блок двигателя"])'}
	kcdo_SK_ON : Tdipar; //диаг. Стопорный клапан открыть//
	{attribute 'export' := '("archive":"True","communication":("cycle":"base"),"journal":"True","name":("full":"диаг. Кран 1 открыть"),"connection":("module":"UE1-A1-DI7-1","type":"НО СК","device_clamp":"UE1","clamp":"Внутр. сигнал"),"subsystem":"Газовая обвязка","group":["Газовая обвязка"])'}
	kcdo_Kr1_ON : Tdipar; //диаг. Кран 1 открыть//
	{attribute 'export' := '("archive":"True","communication":("cycle":"base"),"journal":"True","name":("full":"диаг. Кран 2 открыть"),"connection":("module":"UE1-A1-DI7-2","type":"НО СК","device_clamp":"UE1","clamp":"Внутр. сигнал"),"subsystem":"Газовая обвязка","group":["Газовая обвязка"])'}
	kcdo_Kr2_ON : Tdipar; //диаг. Кран 2 открыть//
	{attribute 'export' := '("archive":"True","communication":("cycle":"base"),"journal":"True","name":("full":"диаг. Кран 4 открыть"),"connection":("module":"UE1-A1-DI7-3","type":"НО СК","device_clamp":"UE1","clamp":"Внутр. сигнал"),"subsystem":"Газовая обвязка","group":["Газовая обвязка"])'}
	kcdo_Kr4_ON : Tdipar; //диаг. Кран 4 открыть//
	{attribute 'export' := '("archive":"True","communication":("cycle":"base"),"journal":"True","name":("full":"диаг. Кран 5 закрыть"),"connection":("module":"UE1-A1-DI7-4","type":"НО СК","device_clamp":"UE1","clamp":"Внутр. сигнал"),"subsystem":"Газовая обвязка","group":["Газовая обвязка"])'}
	kcdo_Kr5_off : Tdipar; //диаг. Кран 5 закрыть//
	{attribute 'export' := '("archive":"True","communication":("cycle":"base"),"journal":"True","name":("full":"диаг. Кран 6 открыть"),"connection":("module":"UE1-A1-DI7-5","type":"НО СК","device_clamp":"UE1","clamp":"Внутр. сигнал"),"subsystem":"Газовая обвязка","group":["Газовая обвязка"])'}
	kcdo_Kr6_ON : Tdipar; //диаг. Кран 6 открыть//
	{attribute 'export' := '("archive":"True","communication":("cycle":"base"),"journal":"True","name":("full":"диаг. Кран 12 открыть (т.г.)"),"connection":("module":"UE1-A1-DI7-6","type":"НО СК","device_clamp":"UE1","clamp":"Внутр. сигнал"),"subsystem":"Газовая обвязка","group":["Газовая обвязка"])'}
	kcdo_Kr12_ON : Tdipar; //диаг. Кран 12 открыть (т.г.)//
	{attribute 'export' := '("archive":"True","communication":("cycle":"base"),"journal":"True","name":("full":"диаг. Кран 11 закрыть (п.г.)"),"connection":("module":"UE1-A1-DI7-8","type":"НО СК","device_clamp":"UE1","clamp":"Внутр. сигнал"),"subsystem":"Газовая обвязка","group":["Газовая обвязка"])'}
	kcdo_Kr11_off : Tdipar; //диаг. Кран 11 закрыть (п.г.)//
	{attribute 'export' := '("archive":"True","communication":("cycle":"base"),"journal":"True","name":("full":"диаг. ЗВУКОВУЮ СИГНАЛИЗАЦИЮ в ГЩУ ВКЛЮЧИТЬ"),"connection":("module":"UE1-A1-DI7-11","type":"НО СК","device_clamp":"UE1","clamp":"Внутр. сигнал"),"subsystem":"Блок автоматики","group":["Блок автоматики"])'}
	kcdo_Sound_ON : Tdipar; //диаг. ЗВУКОВУЮ СИГНАЛИЗАЦИЮ в ГЩУ ВКЛЮЧИТЬ//
	{attribute 'export' := '("archive":"True","communication":("cycle":"base"),"journal":"True","name":("full":"диаг. Эл. магнит управления ВНА включить"),"connection":("module":"UE1-A1-DI7-16","type":"НО СК","device_clamp":"UE1","clamp":"Внутр. сигнал"),"subsystem":"Блок двигателя","group":["Блок двигателя"])'}
	kcdo_VNA_ON : Tdipar; //диаг. Эл. магнит управления ВНА включить//
	{attribute 'export' := '("archive":"True","communication":("cycle":"base"),"journal":"True","name":("full":"диаг. Предохранитель UE1-XTFU1:2 питания модулей DO исправен"),"connection":("module":"UE1-A1-DI7-17","type":"НО СК","device_clamp":"UE1","clamp":"Внутр. сигнал"),"subsystem":"Блок автоматики","group":["Блок автоматики"])'}
	Fuse_DO_UE1 : Tdipar; //диаг. Предохранитель UE1-XTFU1:2 питания модулей DO исправен//
	{attribute 'export' := '("archive":"True","communication":("cycle":"base"),"journal":"True","name":("full":"Перегрузка фильтра EV1 (Осн.)"),"connection":("module":"UPD1-A1-DI1-1","type":"НЗ СК","device_clamp":"UPD1","clamp":"Внутр. сигнал"),"subsystem":"Блок автоматики","group":["Блок автоматики"])'}
	EV1 : Tdipar := (inv := TRUE); //Перегрузка фильтра EV1 (Осн.)//
	{attribute 'export' := '("archive":"True","communication":("cycle":"base"),"journal":"True","name":("full":"Перегрузка фильтра EV2 (Рез.)"),"connection":("module":"UPD1-A1-DI1-2","type":"НЗ СК","device_clamp":"UPD1","clamp":"Внутр. сигнал"),"subsystem":"Блок автоматики","group":["Блок автоматики"])'}
	EV2 : Tdipar := (inv := TRUE); //Перегрузка фильтра EV2 (Рез.)//
	{attribute 'export' := '("archive":"True","communication":("cycle":"base"),"journal":"True","name":("full":"Контроль -AG1"),"connection":("module":"UPD1-A1-DI1-3","type":"НО СК","device_clamp":"UPD1","clamp":"Внутр. сигнал"),"subsystem":"Блок автоматики","group":["Блок автоматики"])'}
	AG1 : Tdipar; //Контроль -AG1//
	{attribute 'export' := '("archive":"True","communication":("cycle":"base"),"journal":"True","name":("full":"Контроль -AG2"),"connection":("module":"UPD1-A1-DI1-4","type":"НО СК","device_clamp":"UPD1","clamp":"Внутр. сигнал"),"subsystem":"Блок автоматики","group":["Блок автоматики"])'}
	AG2 : Tdipar; //Контроль -AG2//
	{attribute 'export' := '("archive":"True","communication":("cycle":"base"),"journal":"True","name":("full":"Контроль -AG5"),"connection":("module":"UPD1-A1-DI1-5","type":"НО СК","device_clamp":"UPD1","clamp":"Внутр. сигнал"),"subsystem":"Блок автоматики","group":["Блок автоматики"])'}
	AG5 : Tdipar; //Контроль -AG5//
	{attribute 'export' := '("archive":"True","communication":("cycle":"base"),"journal":"True","name":("full":"Контроль -AG6"),"connection":("module":"UPD1-A1-DI1-6","type":"НО СК","device_clamp":"UPD1","clamp":"Внутр. сигнал"),"subsystem":"Блок автоматики","group":["Блок автоматики"])'}
	AG6 : Tdipar; //Контроль -AG6//
	{attribute 'export' := '("archive":"True","communication":("cycle":"base"),"journal":"True","name":("full":"Контроль -AG8"),"connection":("module":"UPD1-A1-DI1-7","type":"НО СК","device_clamp":"UPD1","clamp":"Внутр. сигнал"),"subsystem":"Блок автоматики","group":["Блок автоматики"])'}
	AG8 : Tdipar; //Контроль -AG8//
	{attribute 'export' := '("archive":"True","communication":("cycle":"base"),"journal":"True","name":("full":"Контроль -AG9"),"connection":("module":"UPD1-A1-DI1-8","type":"НО СК","device_clamp":"UPD1","clamp":"Внутр. сигнал"),"subsystem":"Блок автоматики","group":["Блок автоматики"])'}
	AG9 : Tdipar; //Контроль -AG9//
	{attribute 'export' := '("archive":"True","communication":("cycle":"base"),"journal":"True","name":("full":"Контроль -AG10"),"connection":("module":"UPD1-A1-DI1-9","type":"НО СК","device_clamp":"UPD1","clamp":"Внутр. сигнал"),"subsystem":"Блок автоматики","group":["Блок автоматики"])'}
	AG10 : Tdipar; //Контроль -AG10//
	{attribute 'export' := '("archive":"True","communication":("cycle":"base"),"journal":"True","name":("full":"Контроль -AG15"),"connection":("module":"UPD1-A1-DI1-10","type":"НО СК","device_clamp":"UPD1","clamp":"Внутр. сигнал"),"subsystem":"Блок автоматики","group":["Блок автоматики"])'}
	AG15 : Tdipar; //Контроль -AG15//
	{attribute 'export' := '("archive":"True","communication":("cycle":"base"),"journal":"True","name":("full":"Контроль -AG16"),"connection":("module":"UPD1-A1-DI1-11","type":"НО СК","device_clamp":"UPD1","clamp":"Внутр. сигнал"),"subsystem":"Блок автоматики","group":["Блок автоматики"])'}
	AG16 : Tdipar; //Контроль -AG16//
	{attribute 'export' := '("archive":"True","communication":("cycle":"base"),"journal":"True","name":("full":"Контроль -AG17"),"connection":("module":"UPD1-A1-DI1-12","type":"НО СК","device_clamp":"UPD1","clamp":"Внутр. сигнал"),"subsystem":"Блок автоматики","group":["Блок автоматики"])'}
	AG17 : Tdipar; //Контроль -AG17//
	{attribute 'export' := '("archive":"True","communication":("cycle":"base"),"journal":"True","name":("full":"Контроль -AG18"),"connection":("module":"UPD1-A1-DI1-13","type":"НО СК","device_clamp":"UPD1","clamp":"Внутр. сигнал"),"subsystem":"Блок автоматики","group":["Блок автоматики"])'}
	AG18 : Tdipar; //Контроль -AG18//
	{attribute 'export' := '("archive":"True","communication":("cycle":"base"),"journal":"True","name":("full":"Ошибка -AUO1"),"connection":("module":"UPD1-A1-DI1-14","type":"НЗ СК","device_clamp":"UPD1","clamp":"Внутр. сигнал"),"subsystem":"Блок автоматики","group":["Блок автоматики"])'}
	Err_AUO1 : Tdipar := (inv := TRUE); //Ошибка -AUO1//
	{attribute 'export' := '("archive":"True","communication":("cycle":"base"),"journal":"True","name":("full":"Контроль основного ввода питания (-KV1)"),"connection":("module":"UPD1-A1-DI2-1","type":"НО СК","device_clamp":"UPD1","clamp":"Внутр. сигнал"),"subsystem":"Блок автоматики","group":["Блок автоматики"])'}
	U_main : Tdipar; //Контроль основного ввода питания (-KV1)//
	{attribute 'export' := '("archive":"True","communication":("cycle":"base"),"journal":"True","name":("full":"Контроль резервного ввода питания (-KV2)"),"connection":("module":"UPD1-A1-DI2-2","type":"НО СК","device_clamp":"UPD1","clamp":"Внутр. сигнал"),"subsystem":"Блок автоматики","group":["Блок автоматики"])'}
	U_res : Tdipar; //Контроль резервного ввода питания (-KV2)//
	{attribute 'export' := '("archive":"True","communication":("cycle":"base"),"journal":"True","name":("full":"Контроль замыкания на землю питания PLC"),"connection":("module":"UPD1-A1-DI2-3","type":"НО СК","device_clamp":"UPD1","clamp":"Внутр. сигнал"),"subsystem":"Блок автоматики","group":["Блок автоматики"])'}
	U_G_PLC : Tdipar; //Контроль замыкания на землю питания PLC//
	{attribute 'export' := '("archive":"True","communication":("cycle":"base"),"journal":"True","name":("full":"Контроль замыкания на землю питания AI"),"connection":("module":"UPD1-A1-DI2-4","type":"НО СК","device_clamp":"UPD1","clamp":"Внутр. сигнал"),"subsystem":"Блок автоматики","group":["Блок автоматики"])'}
	U_G_AI : Tdipar; //Контроль замыкания на землю питания AI//
	{attribute 'export' := '("archive":"True","communication":("cycle":"base"),"journal":"True","name":("full":"Контроль замыкания на землю питания DI"),"connection":("module":"UPD1-A1-DI2-5","type":"НО СК","device_clamp":"UPD1","clamp":"Внутр. сигнал"),"subsystem":"Блок автоматики","group":["Блок автоматики"])'}
	U_G_DI : Tdipar; //Контроль замыкания на землю питания DI//
	{attribute 'export' := '("archive":"True","communication":("cycle":"base"),"journal":"True","name":("full":"Контроль замыкания на FE питания БИЗ"),"connection":("module":"UPD1-A1-DI2-6","type":"НО СК","device_clamp":"UPD1","clamp":"Внутр. сигнал"),"subsystem":"Блок автоматики","group":["Блок автоматики"])'}
	U_G_BIZ : Tdipar; //Контроль замыкания на FE питания БИЗ//
	{attribute 'export' := '("archive":"True","communication":("cycle":"base"),"journal":"True","name":("full":"Контроль замыкания на землю питания ИМ"),"connection":("module":"UPD1-A1-DI2-7","type":"НО СК","device_clamp":"UPD1","clamp":"Внутр. сигнал"),"subsystem":"Блок автоматики","group":["Блок автоматики"])'}
	U_G_AM : Tdipar; //Контроль замыкания на землю питания ИМ//
	{attribute 'export' := '("archive":"True","communication":("cycle":"base"),"journal":"True","name":("full":"Контроль питания AI"),"connection":("module":"UPD1-A1-DI2-8","type":"НО СК","device_clamp":"UPD1","clamp":"Внутр. сигнал"),"subsystem":"Блок автоматики","group":["Блок автоматики"])'}
	U_AI : Tdipar; //Контроль питания AI//
	{attribute 'export' := '("archive":"True","communication":("cycle":"base"),"journal":"True","name":("full":"Контроль питания DI"),"connection":("module":"UPD1-A1-DI2-9","type":"НО СК","device_clamp":"UPD1","clamp":"Внутр. сигнал"),"subsystem":"Блок автоматики","group":["Блок автоматики"])'}
	U_DI : Tdipar; //Контроль питания DI//
	{attribute 'export' := '("archive":"True","communication":("cycle":"base"),"journal":"True","name":("full":"Контроль питания БИЗ"),"connection":("module":"UPD1-A1-DI2-10","type":"НО СК","device_clamp":"UPD1","clamp":"Внутр. сигнал"),"subsystem":"Блок автоматики","group":["Блок автоматики"])'}
	U_BIZ : Tdipar; //Контроль питания БИЗ//
	{attribute 'export' := '("archive":"True","communication":("cycle":"base"),"journal":"True","name":("full":"Контроль питания ИМ"),"connection":("module":"UPD1-A1-DI2-11","type":"НО СК","device_clamp":"UPD1","clamp":"Внутр. сигнал"),"subsystem":"Блок автоматики","group":["Блок автоматики"])'}
	U_AM : Tdipar; //Контроль питания ИМ//
	{attribute 'export' := '("archive":"True","communication":("cycle":"base"),"journal":"True","name":("full":"Контроль питания аппаратуры вибрации, =24 В"),"connection":("module":"UPD1-A1-DI2-12","type":"НО СК","device_clamp":"UPD1","clamp":"Внутр. сигнал"),"subsystem":"Блок автоматики","group":["Блок автоматики"])'}
	Uvs_24 : Tdipar; //Контроль питания аппаратуры вибрации, =24 В//
	{attribute 'export' := '("archive":"True","communication":("cycle":"base"),"journal":"True","name":("full":"Контроль питания дополнительного оборудования, =24В"),"connection":("module":"UPD1-A1-DI2-13","type":"НО СК","device_clamp":"UPD1","clamp":"Внутр. сигнал"),"subsystem":"Блок автоматики","group":["Блок автоматики"])'}
	Uother_24 : Tdipar; //Контроль питания дополнительного оборудования, =24В//
	{attribute 'export' := '("archive":"True","communication":("cycle":"base"),"journal":"True","name":("full":"Контроль питания ИМ2"),"connection":("module":"UPD1-A1-DI2-14","type":"НО СК","device_clamp":"UPD1","clamp":"Внутр. сигнал"),"subsystem":"Блок автоматики","group":["Блок автоматики"])'}
	U_AM2 : Tdipar; //Контроль питания ИМ2//
	{attribute 'export' := '("archive":"True","communication":("cycle":"base"),"journal":"True","name":("full":"Контроль питания ТРК рез."),"connection":("module":"UPD1-A1-DI2-15","type":"НО СК","device_clamp":"UPD1","clamp":"Внутр. сигнал"),"subsystem":"Блок автоматики","group":["Блок автоматики"])'}
	Utrk_res : Tdipar; //Контроль питания ТРК рез.//
	{attribute 'export' := '("archive":"True","communication":("cycle":"base"),"journal":"True","name":("full":"Контроль питания ПРУ"),"connection":("module":"UPD1-A1-DI2-16","type":"НО СК","device_clamp":"UPD1","clamp":"Внутр. сигнал"),"subsystem":"Блок автоматики","group":["Блок автоматики"])'}
	U_PRU : Tdipar; //Контроль питания ПРУ//
	{attribute 'export' := '("archive":"True","communication":("cycle":"base"),"journal":"True","name":("full":"Контроль -AG3"),"connection":("module":"UPD1-A1-DI3-1","type":"НО СК","device_clamp":"UPD1","clamp":"Внутр. сигнал"),"subsystem":"Блок автоматики","group":["Блок автоматики"])'}
	AG3 : Tdipar; //Контроль -AG3//
	{attribute 'export' := '("archive":"True","communication":("cycle":"base"),"journal":"True","name":("full":"Контроль -AG4"),"connection":("module":"UPD1-A1-DI3-2","type":"НО СК","device_clamp":"UPD1","clamp":"Внутр. сигнал"),"subsystem":"Блок автоматики","group":["Блок автоматики"])'}
	AG4 : Tdipar; //Контроль -AG4//
	{attribute 'export' := '("archive":"True","communication":("cycle":"base"),"journal":"True","name":("full":"Контроль питания ТРК осн."),"connection":("module":"UPD1-A1-DI3-3","type":"НО СК","device_clamp":"UPD1","clamp":"Внутр. сигнал"),"subsystem":"Блок автоматики","group":["Блок автоматики"])'}
	Utrk_main : Tdipar; //Контроль питания ТРК осн.//
	{attribute 'export' := '("archive":"True","communication":("cycle":"base"),"journal":"True","name":("full":"БЭО. Перегрузка фильтра EV3 (Осн. БЭО)"),"connection":("module":"UPD1-A1-DI3-5","type":"НЗ СК","device_clamp":"UPD1","clamp":"Внутр. сигнал"),"subsystem":"Блок автоматики","group":["Блок автоматики"])'}
	EV3 : Tdipar := (inv := TRUE); //БЭО. Перегрузка фильтра EV3 (Осн. БЭО)//
	{attribute 'export' := '("archive":"True","communication":("cycle":"base"),"journal":"True","name":("full":"БЭО. Перегрузка фильтра EV4 (Рез. БЭО)"),"connection":("module":"UPD1-A1-DI3-6","type":"НЗ СК","device_clamp":"UPD1","clamp":"Внутр. сигнал"),"subsystem":"Блок автоматики","group":["Блок автоматики"])'}
	EV4 : Tdipar := (inv := TRUE); //БЭО. Перегрузка фильтра EV4 (Рез. БЭО)//
	{attribute 'export' := '("archive":"True","communication":("cycle":"base"),"journal":"True","name":("full":"БЭО. Контроль основного ввода питания БЭО (-KV3)"),"connection":("module":"UPD1-A1-DI3-7","type":"НО СК","device_clamp":"UPD1","clamp":"Внутр. сигнал"),"subsystem":"Блок автоматики","group":["Блок автоматики"])'}
	Ubeo_main : Tdipar; //БЭО. Контроль основного ввода питания БЭО (-KV3)//
	{attribute 'export' := '("archive":"True","communication":("cycle":"base"),"journal":"True","name":("full":"БЭО. Контроль резервного ввода питания БЭО (-KV4)"),"connection":("module":"UPD1-A1-DI3-8","type":"НО СК","device_clamp":"UPD1","clamp":"Внутр. сигнал"),"subsystem":"Блок автоматики","group":["Блок автоматики"])'}
	Ubeo_res : Tdipar; //БЭО. Контроль резервного ввода питания БЭО (-KV4)//
	{attribute 'export' := '("archive":"True","communication":("cycle":"base"),"journal":"True","name":("full":"БЭО. Контроль -AG11"),"connection":("module":"UPD1-A1-DI3-9","type":"НО СК","device_clamp":"UPD1","clamp":"Внутр. сигнал"),"subsystem":"Блок автоматики","group":["Блок автоматики"])'}
	AG11 : Tdipar; //БЭО. Контроль -AG11//
	{attribute 'export' := '("archive":"True","communication":("cycle":"base"),"journal":"True","name":("full":"БЭО. Контроль -AG12"),"connection":("module":"UPD1-A1-DI3-10","type":"НО СК","device_clamp":"UPD1","clamp":"Внутр. сигнал"),"subsystem":"Блок автоматики","group":["Блок автоматики"])'}
	AG12 : Tdipar; //БЭО. Контроль -AG12//
	{attribute 'export' := '("archive":"True","communication":("cycle":"base"),"journal":"True","name":("full":"БЭО. Контроль замыкания на землю питания БЭО (-KR5)"),"connection":("module":"UPD1-A1-DI3-11","type":"НО СК","device_clamp":"UPD1","clamp":"Внутр. сигнал"),"subsystem":"Блок автоматики","group":["Блок автоматики"])'}
	U_G_KR5 : Tdipar; //БЭО. Контроль замыкания на землю питания БЭО (-KR5)//
	{attribute 'export' := '("archive":"True","communication":("cycle":"base"),"journal":"True","name":("full":"БЭО. Контроль питания кн. ЭАО"),"connection":("module":"UPD1-A1-DI3-12","type":"НО СК","device_clamp":"UPD1","clamp":"Внутр. сигнал"),"subsystem":"Блок автоматики","group":["Блок автоматики"])'}
	U_KEAO : Tdipar; //БЭО. Контроль питания кн. ЭАО//
	{attribute 'export' := '("archive":"True","communication":("cycle":"base"),"journal":"True","name":("full":"БЭО. Контроль питания БЭО"),"connection":("module":"UPD1-A1-DI3-13","type":"НО СК","device_clamp":"UPD1","clamp":"Внутр. сигнал"),"subsystem":"Блок автоматики","group":["Блок автоматики"])'}
	U_BEO : Tdipar; //БЭО. Контроль питания БЭО//
	{attribute 'export' := '("archive":"True","communication":("cycle":"base"),"journal":"True","name":("full":"БЭО. Контроль питания БЗА"),"connection":("module":"UPD1-A1-DI3-14","type":"НО СК","device_clamp":"UPD1","clamp":"Внутр. сигнал"),"subsystem":"Блок автоматики","group":["Блок автоматики"])'}
	U_BZA : Tdipar; //БЭО. Контроль питания БЗА//
END_VAR
(* global variable list dopar *)
{region INFO}
(*
 Назначение: Используется для хранения, инициализации и передачи на ВУ значений и состояния выходных дискретных параметров
 Автор:      /Andrey/ 16.07.2025 17:15:05
 Версия ТЭ5: v00.00.01
 Проект:     KA107
*)
{endregion}
{attribute 'qualified_only'}
{attribute 'symbol' := 'readwrite'}
VAR_GLOBAL
	{attribute 'symbol' := 'none'}
	common : Tdopar;
	{attribute 'export' := '("archive":"True","communication":("cycle":"base"),"journal":"True","name":("full":"Включить вытяжной Вент.ВОУ"),"connection":("module":"UCP1-A2-DO1-17","type":"НО СК","device_clamp":"UCP1","clamp":"XDO2:1A XDO2:1B"),"subsystem":"Блок автоматики","group":["Блок автоматики"])'}
	VV_VOU_ON : Tdopar := (kc_type := 0); //Включить вытяжной Вент.ВОУ//
	{attribute 'export' := '("archive":"True","communication":("cycle":"base"),"journal":"True","name":("full":"Отключить вытяжной Вент.ВОУ"),"connection":("module":"UCP1-A2-DO1-18","type":"НЗ СК","device_clamp":"UCP1","clamp":"XDO2:2A XDO2:2B"),"subsystem":"Блок автоматики","group":["Блок автоматики"])'}
	VV_VOU_OFF : Tdopar := (kc_type := 0); //Отключить вытяжной Вент.ВОУ//
	{attribute 'export' := '("archive":"True","communication":("cycle":"base"),"journal":"True","name":("full":"Вентилятор 1 маслоохладителей АВОМ включить"),"connection":("module":"UCP1-A2-DO1-19","type":"НО СК","device_clamp":"UCP1","clamp":"XDO2:3A XDO2:3B"),"subsystem":"АВОМ","group":["АВОМ"])'}
	Vn1_AVOM_ON : Tdopar := (kc_type := 0); //Вентилятор 1 маслоохладителей АВОМ включить//
	{attribute 'export' := '("archive":"True","communication":("cycle":"base"),"journal":"True","name":("full":"Вентилятор 1 маслоохладителей АВОМ отключить"),"connection":("module":"UCP1-A2-DO1-20","type":"НЗ СК","device_clamp":"UCP1","clamp":"XDO2:4A XDO2:4B"),"subsystem":"АВОМ","group":["АВОМ"])'}
	Vn1_AVOM_OFF : Tdopar := (kc_type := 0); //Вентилятор 1 маслоохладителей АВОМ отключить//
	{attribute 'export' := '("archive":"True","communication":("cycle":"base"),"journal":"True","name":("full":"Вентилятор 2 маслоохладителей АВОМ включить"),"connection":("module":"UCP1-A2-DO1-21","type":"НО СК","device_clamp":"UCP1","clamp":"XDO2:5A XDO2:5B"),"subsystem":"АВОМ","group":["АВОМ"])'}
	Vn2_AVOM_ON : Tdopar := (kc_type := 0); //Вентилятор 2 маслоохладителей АВОМ включить//
	{attribute 'export' := '("archive":"True","communication":("cycle":"base"),"journal":"True","name":("full":"Вентилятор 2 маслоохладителей АВОМ отключить"),"connection":("module":"UCP1-A2-DO1-22","type":"НЗ СК","device_clamp":"UCP1","clamp":"XDO2:6A XDO2:6B"),"subsystem":"АВОМ","group":["АВОМ"])'}
	Vn2_AVOM_OFF : Tdopar := (kc_type := 0); //Вентилятор 2 маслоохладителей АВОМ отключить//
	{attribute 'export' := '("archive":"True","communication":("cycle":"base"),"journal":"True","name":("full":"Вентилятор 3 маслоохладителей АВОМ включить"),"connection":("module":"UCP1-A2-DO1-23","type":"НО СК","device_clamp":"UCP1","clamp":"XDO2:7A XDO2:7B"),"subsystem":"АВОМ","group":["АВОМ"])'}
	Vn3_AVOM_ON : Tdopar := (kc_type := 0); //Вентилятор 3 маслоохладителей АВОМ включить//
	{attribute 'export' := '("archive":"True","communication":("cycle":"base"),"journal":"True","name":("full":"Вентилятор 3 маслоохладителей АВОМ отключить"),"connection":("module":"UCP1-A2-DO1-24","type":"НЗ СК","device_clamp":"UCP1","clamp":"XDO2:8A XDO2:8B"),"subsystem":"АВОМ","group":["АВОМ"])'}
	Vn3_AVOM_OFF : Tdopar := (kc_type := 0); //Вентилятор 3 маслоохладителей АВОМ отключить//
	{attribute 'export' := '("archive":"True","communication":("cycle":"base"),"journal":"True","name":("full":"Вентилятор 4 маслоохладителей АВОМ включить"),"connection":("module":"UCP1-A2-DO1-25","type":"НО СК","device_clamp":"UCP1","clamp":"XDO2:9A XDO2:9B"),"subsystem":"АВОМ","group":["АВОМ"])'}
	Vn4_AVOM_ON : Tdopar := (kc_type := 0); //Вентилятор 4 маслоохладителей АВОМ включить//
	{attribute 'export' := '("archive":"True","communication":("cycle":"base"),"journal":"True","name":("full":"Вентилятор 4 маслоохладителей АВОМ отключить"),"connection":("module":"UCP1-A2-DO1-26","type":"НЗ СК","device_clamp":"UCP1","clamp":"XDO2:10A XDO2:10B"),"subsystem":"АВОМ","group":["АВОМ"])'}
	Vn4_AVOM_OFF : Tdopar := (kc_type := 0); //Вентилятор 4 маслоохладителей АВОМ отключить//
	{attribute 'export' := '("archive":"True","communication":("cycle":"base"),"journal":"True","name":("full":"Вытяжной вентилятор нагнетателя ВВН включить"),"connection":("module":"UCP1-A2-DO1-27","type":"НО СК","device_clamp":"UCP1","clamp":"XDO2:11A XDO2:11B"),"subsystem":"Блок автоматики","group":["Блок автоматики"])'}
	VVN_ON : Tdopar := (kc_type := 0); //Вытяжной вентилятор нагнетателя ВВН включить//
	{attribute 'export' := '("archive":"True","communication":("cycle":"base"),"journal":"True","name":("full":"Вытяжной вентилятор нагнетателя ВВН отключить"),"connection":("module":"UCP1-A2-DO1-28","type":"НЗ СК","device_clamp":"UCP1","clamp":"XDO2:12A XDO2:12B"),"subsystem":"Блок автоматики","group":["Блок автоматики"])'}
	VVN_OFF : Tdopar := (kc_type := 0); //Вытяжной вентилятор нагнетателя ВВН отключить//
	{attribute 'export' := '("archive":"True","communication":("cycle":"base"),"journal":"True","name":("full":"Пусковой насос уплотнения отключить"),"connection":("module":"UCP1-A2-DO1-31","type":"НЗ СК","device_clamp":"UCP1","clamp":"XDO2:15A XDO2:15B"),"subsystem":"Маслосистема К","group":["Маслосистема К"])'}
	PNU_OFF : Tdopar := (kc_type := 0); //Пусковой насос уплотнения отключить//
	{attribute 'export' := '("archive":"True","communication":("cycle":"base"),"journal":"True","name":("full":"Пусковой насос смазки отключить"),"connection":("module":"UCP1-A2-DO1-32","type":"НЗ СК","device_clamp":"UCP1","clamp":"XDO2:16A XDO2:16B"),"subsystem":"Маслосистема Д","group":["Маслосистема Д"])'}
	PNS_OFF : Tdopar := (kc_type := 0); //Пусковой насос смазки отключить//
	{attribute 'export' := '("archive":"True","communication":("cycle":"base"),"journal":"True","name":("full":"Кран 1 закрыть"),"connection":("module":"UE1-A1-DO1-1","type":"U","device_clamp":"UE1","clamp":"XDO1:1A XDO1:1B"),"subsystem":"Газовая обвязка","group":["Газовая обвязка"])'}
	Kr1_OFF : Tdopar := (kc_type := 1); //Кран 1 закрыть//
	{attribute 'export' := '("archive":"True","communication":("cycle":"base"),"journal":"True","name":("full":"Кран 1 смазка"),"connection":("module":"UE1-A1-DO1-2","type":"U","device_clamp":"UE1","clamp":"XDO1:2A XDO1:2B"),"subsystem":"Газовая обвязка","group":["Газовая обвязка"])'}
	Kr1m_ON : Tdopar := (kc_type := 1); //Кран 1 смазка//
	{attribute 'export' := '("archive":"True","communication":("cycle":"base"),"journal":"True","name":("full":"Кран 2 закрыть"),"connection":("module":"UE1-A1-DO1-3","type":"U","device_clamp":"UE1","clamp":"XDO1:3A XDO1:3B"),"subsystem":"Газовая обвязка","group":["Газовая обвязка"])'}
	Kr2_OFF : Tdopar := (kc_type := 1); //Кран 2 закрыть//
	{attribute 'export' := '("archive":"True","communication":("cycle":"base"),"journal":"True","name":("full":"Кран 2 смазка"),"connection":("module":"UE1-A1-DO1-4","type":"U","device_clamp":"UE1","clamp":"XDO1:4A XDO1:4B"),"subsystem":"Газовая обвязка","group":["Газовая обвязка"])'}
	Kr2m_ON : Tdopar := (kc_type := 1); //Кран 2 смазка//
	{attribute 'export' := '("archive":"True","communication":("cycle":"base"),"journal":"True","name":("full":"Кран 4 закрыть"),"connection":("module":"UE1-A1-DO1-5","type":"U","device_clamp":"UE1","clamp":"XDO1:5A XDO1:5B"),"subsystem":"Газовая обвязка","group":["Газовая обвязка"])'}
	Kr4_OFF : Tdopar := (kc_type := 1); //Кран 4 закрыть//
	{attribute 'export' := '("archive":"True","communication":("cycle":"base"),"journal":"True","name":("full":"Кран 5 открыть"),"connection":("module":"UE1-A1-DO1-7","type":"U","device_clamp":"UE1","clamp":"XDO1:7A XDO1:7B"),"subsystem":"Газовая обвязка","group":["Газовая обвязка"])'}
	Kr5_ON : Tdopar := (kc_type := 1); //Кран 5 открыть//
	{attribute 'export' := '("archive":"True","communication":("cycle":"base"),"journal":"True","name":("full":"Кран 6 закрыть"),"connection":("module":"UE1-A1-DO1-9","type":"U","device_clamp":"UE1","clamp":"XDO1:9A XDO1:9B"),"subsystem":"Газовая обвязка","group":["Газовая обвязка"])'}
	Kr6_OFF : Tdopar := (kc_type := 1); //Кран 6 закрыть//
	{attribute 'export' := '("archive":"True","communication":("cycle":"base"),"journal":"True","name":("full":"Кран 6 смазка"),"connection":("module":"UE1-A1-DO1-10","type":"U","device_clamp":"UE1","clamp":"XDO1:10A XDO1:10B"),"subsystem":"Газовая обвязка","group":["Газовая обвязка"])'}
	Kr6m_ON : Tdopar := (kc_type := 1); //Кран 6 смазка//
	{attribute 'export' := '("archive":"True","communication":("cycle":"base"),"journal":"True","name":("full":"Кран 12 закрыть (т.г.), кран 9 (т.г. свеч.) открыть"),"connection":("module":"UE1-A1-DO1-11","type":"U","device_clamp":"UE1","clamp":"XDO1:11A XDO1:11B"),"subsystem":"Газовая обвязка","group":["Газовая обвязка"])'}
	KR12_OFF : Tdopar := (kc_type := 1); //Кран 12 закрыть (т.г.), кран 9 (т.г. свеч.) открыть//
	{attribute 'export' := '("archive":"True","communication":("cycle":"base"),"journal":"True","name":("full":"Кран 11 открыть (п.г.) кран 10(п.г.свеч.) закрыть"),"connection":("module":"UE1-A1-DO1-15","type":"U","device_clamp":"UE1","clamp":"XDO1:15A XDO1:15B"),"subsystem":"Газовая обвязка","group":["Газовая обвязка"])'}
	Kr11_ON : Tdopar := (kc_type := 1); //Кран 11 открыть (п.г.) кран 10(п.г.свеч.) закрыть//
	{attribute 'export' := '("archive":"True","communication":("cycle":"base"),"journal":"True","name":("full":"Включение КПВ 1,5"),"connection":("module":"UE1-A1-DO1-19","type":"U","device_clamp":"UE1","clamp":"XDO1:19A XDO1:19B"),"subsystem":"Блок двигателя","group":["Блок двигателя"])'}
	KPV15_ON : Tdopar := (kc_type := 1); //Включение КПВ 1,5//
	{attribute 'export' := '("archive":"True","communication":("cycle":"base"),"journal":"True","name":("full":"Включение КПВ 2,3"),"connection":("module":"UE1-A1-DO1-20","type":"U","device_clamp":"UE1","clamp":"XDO1:20A XDO1:20B"),"subsystem":"Блок двигателя","group":["Блок двигателя"])'}
	KPV23_OFF : Tdopar := (kc_type := 1); //Включение КПВ 2,3//
	{attribute 'export' := '("archive":"True","communication":("cycle":"base"),"journal":"True","name":("full":"Включение КПВ 4"),"connection":("module":"UE1-A1-DO1-21","type":"U","device_clamp":"UE1","clamp":"XDO1:21A XDO1:21B"),"subsystem":"Блок двигателя","group":["Блок двигателя"])'}
	KPV4_OFF : Tdopar := (kc_type := 1); //Включение КПВ 4//
	{attribute 'export' := '("archive":"True","communication":("cycle":"fast"),"journal":"True","name":("full":"Стопорный клапан открыть"),"connection":("module":"UE1-A1-DO1-22","type":"U","device_clamp":"UE1","clamp":"XDO1:22A XDO1:22B"),"subsystem":"Блок топливного газа","group":["Блок топливного газа"])'}
	SK_ON : Tdopar := (kc_type := 1); //Стопорный клапан открыть//
	{attribute 'export' := '("archive":"True","communication":("cycle":"base"),"journal":"True","name":("full":"Пусковой насос смазки включить"),"connection":("module":"UE1-A1-DO1-30","type":"НО СК","device_clamp":"UE1","clamp":"XDO1:30A XDO1:30B"),"subsystem":"Маслосистема Д","group":["Маслосистема Д"])'}
	PNS_ON : Tdopar := (kc_type := 0); //Пусковой насос смазки включить//
	{attribute 'export' := '("archive":"True","communication":("cycle":"base"),"journal":"True","name":("full":"Пусковой насос уплотнения включить"),"connection":("module":"UE1-A1-DO1-31","type":"НО СК","device_clamp":"UE1","clamp":"XDO1:31A XDO1:31B"),"subsystem":"Маслосистема К","group":["Маслосистема К"])'}
	PNU_ON : Tdopar := (kc_type := 0); //Пусковой насос уплотнения включить//
	{attribute 'export' := '("archive":"True","communication":("cycle":"base"),"journal":"False","name":("full":"БЭО. Работа-1"),"connection":("module":"UE1-A1-DO1-32","type":"U","device_clamp":"UE1","clamp":"Внутр. сигнал"),"subsystem":"Блок автоматики","group":["Блок автоматики"])'}
	BEO_w1 : Tdopar := (kc_type := 0); //БЭО. Работа-1//
	{attribute 'export' := '("archive":"True","communication":("cycle":"base"),"journal":"True","name":("full":"Кран 1 открыть"),"connection":("module":"UE1-A1-DO2-1","type":"U","device_clamp":"UE1","clamp":"XDO2:1A XDO2:1B"),"subsystem":"Газовая обвязка","group":["Газовая обвязка"])'}
	Kr1_ON : Tdopar := (kc_type := 1); //Кран 1 открыть//
	{attribute 'export' := '("archive":"True","communication":("cycle":"base"),"journal":"True","name":("full":"Кран 2 открыть"),"connection":("module":"UE1-A1-DO2-2","type":"U","device_clamp":"UE1","clamp":"XDO2:2A XDO2:2B"),"subsystem":"Газовая обвязка","group":["Газовая обвязка"])'}
	Kr2_ON : Tdopar := (kc_type := 1); //Кран 2 открыть//
	{attribute 'export' := '("archive":"True","communication":("cycle":"base"),"journal":"True","name":("full":"Кран 4 открыть"),"connection":("module":"UE1-A1-DO2-3","type":"U","device_clamp":"UE1","clamp":"XDO2:3A XDO2:3B"),"subsystem":"Газовая обвязка","group":["Газовая обвязка"])'}
	Kr4_ON : Tdopar := (kc_type := 1); //Кран 4 открыть//
	{attribute 'export' := '("archive":"True","communication":("cycle":"base"),"journal":"True","name":("full":"Кран 5 закрыть"),"connection":("module":"UE1-A1-DO2-4","type":"U","device_clamp":"UE1","clamp":"XDO2:4A XDO2:4B"),"subsystem":"Газовая обвязка","group":["Газовая обвязка"])'}
	Kr5_OFF : Tdopar := (kc_type := 1); //Кран 5 закрыть//
	{attribute 'export' := '("archive":"True","communication":("cycle":"base"),"journal":"True","name":("full":"Кран 6 открыть"),"connection":("module":"UE1-A1-DO2-5","type":"U","device_clamp":"UE1","clamp":"XDO2:5A XDO2:5B"),"subsystem":"Газовая обвязка","group":["Газовая обвязка"])'}
	Kr6_ON : Tdopar := (kc_type := 1); //Кран 6 открыть//
	{attribute 'export' := '("archive":"True","communication":("cycle":"base"),"journal":"True","name":("full":"Кран 12 открыть (т.г.), кран 9 (т.г. свеч.) закрыть"),"connection":("module":"UE1-A1-DO2-6","type":"U","device_clamp":"UE1","clamp":"XDO2:6A XDO2:6B"),"subsystem":"Газовая обвязка","group":["Газовая обвязка"])'}
	Kr12_ON : Tdopar := (kc_type := 1); //Кран 12 открыть (т.г.), кран 9 (т.г. свеч.) закрыть//
	{attribute 'export' := '("archive":"True","communication":("cycle":"base"),"journal":"True","name":("full":"Кран 11 закрыть (п.г.) Кран 10(п.г.свеч.) открыть"),"connection":("module":"UE1-A1-DO2-8","type":"U","device_clamp":"UE1","clamp":"XDO2:8A XDO2:8B"),"subsystem":"Газовая обвязка","group":["Газовая обвязка"])'}
	Kr11_OFF : Tdopar := (kc_type := 1); //Кран 11 закрыть (п.г.) Кран 10(п.г.свеч.) открыть//
	{attribute 'export' := '("archive":"True","communication":("cycle":"base"),"journal":"True","name":("full":"ЗВУКОВУЮ СИГНАЛИЗАЦИЮ в ГЩУ ВКЛЮЧИТЬ"),"connection":("module":"UE1-A1-DO2-11","type":"U","device_clamp":"UE1","clamp":"XDO2:11A XDO2:11B"),"subsystem":"Блок автоматики","group":["Блок автоматики"])'}
	Sound_ON : Tdopar := (kc_type := 1); //ЗВУКОВУЮ СИГНАЛИЗАЦИЮ в ГЩУ ВКЛЮЧИТЬ//
	{attribute 'export' := '("archive":"True","communication":("cycle":"base"),"journal":"True","name":("full":"Эл. магнит управления ВНА включить"),"connection":("module":"UE1-A1-DO2-16","type":"U","device_clamp":"UE1","clamp":"XDO2:16A XDO2:16B"),"subsystem":"Блок двигателя","group":["Блок двигателя"])'}
	VNA_ON : Tdopar := (kc_type := 1); //Эл. магнит управления ВНА включить//
	{attribute 'export' := '("archive":"True","communication":("cycle":"base"),"journal":"True","name":("full":"Включить агрегат зажигания"),"connection":("module":"UE1-A1-DO2-18","type":"U","device_clamp":"UE1","clamp":"XDO2:18A XDO2:18B"),"subsystem":"Блок двигателя","group":["Блок двигателя"])'}
	AZ_ON : Tdopar := (kc_type := 0); //Включить агрегат зажигания//
	{attribute 'export' := '("archive":"True","communication":("cycle":"base"),"journal":"True","name":("full":"Обогрев ВНА включить"),"connection":("module":"UE1-A1-DO2-19","type":"U","device_clamp":"UE1","clamp":"XDO2:19A XDO2:19B"),"subsystem":"Блок двигателя","group":["Блок двигателя"])'}
	VNA_heat_ON : Tdopar := (kc_type := 0); //Обогрев ВНА включить//
	{attribute 'export' := '("archive":"True","communication":("cycle":"base"),"journal":"True","name":("full":"Кран 13 открыть (заслонка возд. стартера)"),"connection":("module":"UE1-A1-DO2-22","type":"U","clamp":"XDO2:22A XDO2:22B"),"subsystem":"Газовая обвязка","group":["Газовая обвязка"])'}
	Kr13_ON : Tdopar := (kc_type := 0); //Кран 13 открыть (заслонка возд. стартера)//
	{attribute 'export' := '("archive":"True","communication":("cycle":"base"),"journal":"True","name":("full":"Кран 15 открыть"),"connection":("module":"UE1-A1-DO2-23","type":"U","device_clamp":"UE1","clamp":"XDO2:23A XDO2:23B"),"subsystem":"Газовая обвязка","group":["Газовая обвязка"])'}
	Kr15_ON : Tdopar := (kc_type := 0); //Кран 15 открыть//
	{attribute 'export' := '("archive":"True","communication":("cycle":"base"),"journal":"True","name":("full":"Контроль ИВ-Д-ПФ-1М.3Н.1-01"),"connection":("module":"UE1-A1-DO2-29","type":"U","device_clamp":"UE1","clamp":"XDO2:29A"),"subsystem":"Блок автоматики","group":["Блок автоматики"])'}
	Vibr_ctrl : Tdopar := (kc_type := 0); //Контроль ИВ-Д-ПФ-1М.3Н.1-01//
	{attribute 'export' := '("archive":"True","communication":("cycle":"base"),"journal":"True","name":("full":"Контроль БЗА"),"connection":("module":"UE1-A1-DO2-30","type":"НО СК","device_clamp":"UE1","clamp":"Внутр. сигнал"),"subsystem":"Блок автоматики","group":["Блок автоматики"])'}
	BZA_ctrl : Tdopar := (kc_type := 0); //Контроль БЗА//
	{attribute 'export' := '("archive":"True","communication":("cycle":"base"),"journal":"True","name":("full":"Сброс БЗА"),"connection":("module":"UE1-A1-DO2-31","type":"НО СК","device_clamp":"UE1","clamp":"Внутр. сигнал"),"subsystem":"Блок автоматики","group":["Блок автоматики"])'}
	BZA_reset : Tdopar := (kc_type := 0); //Сброс БЗА//
	{attribute 'export' := '("archive":"True","communication":("cycle":"base"),"journal":"False","name":("full":"БЭО. Работа-2"),"connection":("module":"UE1-A1-DO2-32","type":"U","device_clamp":"UE1","clamp":"Внутр. сигнал"),"subsystem":"Блок автоматики","group":["Блок автоматики"])'}
	BEO_w2 : Tdopar := (kc_type := 0); //БЭО. Работа-2//
END_VAR
(* global variable list check *)
{attribute 'qualified_only' := ''}
{attribute 'symbol' := 'none'}
VAR_GLOBAL
	tmr12H		: TON 	:= (PT := TIME#720M0S0MS);	// Отсчёт 12 часов 
	tmrImit		: TON 	:= (PT := TIME#5S0MS);		// таймер для имитатора
	tmrCancelPrm: TON	:= (PT := TIME#11S0MS);		// запрет кнопки Отмена
	prm_start: BOOL;
	ReadytoSF: BOOL;
	ready: ENUM_ReadyToStart;
	btn: BOOL;
END_VAR
(* global variable list tch *)
///
/// Назначение:   Используется для хранения, инициализации и передачи на ВУ технологических сигнализаций
/// Автор:        /Chekmarev/ 18.03.2025
/// Проект:       KA107
{attribute 'qualified_only' := ''}
{attribute 'symbol' := 'read'}
VAR_GLOBAL
	Unlock			: Ttch; // Деблокировка
	nGas_N			: Ttch; // Нет газа в контуре компрессора
	Gas_N			: Ttch; // Газ в контуре компрессора
	ReadyHP			: Ttch; // Готов к ХП
	ReadyKPK		: Ttch; // Готов к КПК
	ReadyAPK		: Ttch; // Готов к АПК
	ReadyPZ			: Ttch; // Готов к ПЗ
	PrepareStart	: Ttch; // Подготовка к пуску
	Check_SAU		: Ttch; // Контроль САУ
	GTDstart		: Ttch; // Запуск двигателя
	GTDwork			: Ttch; // Агрегат работает
	GTDHeat			: Ttch; // Прогрев двигателя
	GTDcool			: Ttch; // Охлаждение двигателя
	CheckAlarm_on 	: Ttch; // Запущен режим проверки защит
  	AS_antisurgeBrk : Ttch; // Отказ антипомпажной защиты
  	AS_mainContBrk 	: Ttch; // Отказ основного контура вычисления помпажного запаса
  	AS_res1ContBrk 	: Ttch; // Отказ 1 резервного контура вычисления помпажного запаса
  	AS_res2ContBrk 	: Ttch; // Отказ 2 резервного контура вычисления помпажного запаса
  	AS_preSurge 		: Ttch; // сигнал "Предпомпажное состояние"
  	AS_surge 			: Ttch; // сигнал "Помпаж нагнетателя"
  	AS_surgeAlertBrk 	: Ttch; // сигнал "Отказ сигнализатора помпажа"
  	AS_surgeSign_ddPconf : Ttch; // внутренний сигнал "Предпомпажное состояние" по падению dP на конфузоре //Dergaev 2024-11-02
  	AS_surgeSign_dNst 	: Ttch; // внутренний сигнал "Предпомпажное состояние" по росту частоты вращения  //Dergaev 2024-11-02
	
END_VAR
(* global variable list alg *)
///
/// Назначение:   Используется для хранения внутренних алгоритмических сигналов
/// Автор:        /Chekmarev/ 18.02.2025
/// Проект:       KA107
{attribute 'qualified_only' := ''}
{attribute 'symbol' := 'none'}
VAR_GLOBAL
	/// Состояния
	V_000	: BOOL;
	work	: BOOL;
	start	: BOOL;
	stop	: BOOL;
	AO		: BOOL;
	AO_old	: BOOL;
	AOss	: BOOL;
	AObs	: BOOL;
	NO		: BOOL;
	reserve	: BOOL;
	test	: BOOL;
	// Прирост давления в контуре > 0.05 МПа в секунду 
	nIncPgN	: BOOL;
	// Защита по маслосистеме нагнетателя
	sh_PmN	: BOOL;
	// Защита по маслосистеме ТК и СТ
	sh_PmGTD: BOOL;
	// Защита по ТГ
	sh_TG	: BOOL;
	// Защита по давлению масла перед ДГ (САР)
	sh_SAR	: BOOL;
	// Защита по перепаду "масло-газ"
	sh_dPmg	: BOOL;
	// Защита по не розжигу
	sh_nIgnition: BOOL;
	// Защита по нераскрутке на старте
	sh_nBoost	: BOOL;
	// Контроль защит
	sh_cntrl	: BOOL;
	
	KPV234_wOpen: BOOL;
	// Защита по незарытию КПВ1,5
	KPV15_wOpen	: BOOL;
	// Защита по неоткрытию КПВ1,5
	KPV15_nOpen	: BOOL;
	// Нормальный останов из последовательностей в ТР
	normalStopCom: BOOL;
	// Аварийный останов из последовательностей в ТР
	emergStopCom: BOOL;
	// Управление ВНА из последовательностей
	//VNA_on		: BOOL;
	// Количество работоспособных термопар перед СТ
	TstInWork	: BYTE;
	// Защита по маслосистеме воздушного стартера
	sh_Starter	: BOOL;
	// Защита по давлению газа перед краном 13
	sh_Pg_inKR13: BOOL;
	// Закрытие крана 6 по снятию s_tunpar.ASprot.emergOpenBypass
	KR6_off_after_emergOpenBypass : TEdgeDetect;
	
	AObs_tech	: BOOL;
	AOss_tech	: BOOL;
	VOss_tech	: BOOL;
END_VAR
(* global variable list imitGPA *)
{attribute 'qualified_only' := ''}
VAR_GLOBAL
	///tau			: REAL;	
	imit_start: R_TRIG;
	init: BOOL;
	imit_on: BOOL;
END_VAR
(* global variable list GVL *)
{attribute 'symbol' := 'none'}
VAR_GLOBAL
	// Режимы
	{attribute 'symbol' := 'read'}
	mde_hmi: Tmde_hmi;
	
	// Наработка агрегата
	{attribute 'symbol' := 'readwrite'}
	MotoClockGPA	: TMotoClockHandler; 
	
	{attribute 'symbol' := 'none'}
	Pg_inN_old: REAL;
END_VAR
(* global variable list GVL_IMIT *)
{attribute 'qualified_only' := ''}
VAR_GLOBAL
	imitTuns: TImitEngineTuns := (openToGt := (nPoint := 4, point := [(x := REAL#0, y := REAL#0), (x := REAL#25, y := REAL#573),(x := REAL#50, y := REAL#1368), (x := REAL#100, y := REAL#3727)]), 
		GtToNvd := (nPoint := 3, point := [(x := REAL#0, y := REAL#0), (x := REAL#1986, y := REAL#8200), (x := REAL#3000, y := REAL#10000)]), 
		GtToTst := (nPoint := 4, point := [(x := REAL#0, y := REAL#0), (x := REAL#200, y := REAL#300), (x := REAL#1300, y := REAL#400), (x := REAL#3000, y := REAL#800)]), 
		NvdToTauNvd := (nPoint := 5, point := [(x := REAL#0, y := REAL#20), (x := REAL#2000, y := REAL#10), (x := REAL#4500, y := REAL#5), (x := REAL#6300, y := REAL#1), (x := REAL#10000, y := REAL#0.5)]), 
		NvdToTauTst := (nPoint := 2, point := [(x := REAL#0, y := REAL#1), (x := REAL#10000, y := REAL#0.2)]), 
		NvdToTauPk := (nPoint := 2, point := [(x := REAL#0, y := REAL#2), (x := REAL#10000, y := REAL#0.7)]), 
		NstToTauNst := (nPoint := 2, point := [(x := REAL#0, y := REAL#2), (x := REAL#10000, y := REAL#1)]), 
		NvdToTst := (nPoint := 2, point := [(x := REAL#0, y := REAL#10), (x := REAL#10000, y := REAL#200)]), 
		NvdToPk := (nPoint := 2, point := [(x := REAL#0, y := REAL#0), (x := REAL#10000, y := REAL#1.4)]), 
		NvdToNst := (nPoint := 3, point := [(x := REAL#0, y := REAL#0), (x := REAL#2000, y := REAL#0), (x := REAL#10000, y := REAL#10000)]), 
		DUSdz := 0.05, 
		DUSrate := 300, 
		NvdStart := 2100);
	starter: BOOL;
	imitEngine: TEngineModel := (cycle := REAL#0.04, SDpresent := FALSE, NDpresent := FALSE, PkPresent := TRUE, DUSaddPresent := FALSE, elStart := FALSE, step := (cycle_time_fast / 5));
END_VAR
(* global variable list s_aspar *)
///
/// Назначение: 		Используется для хранения и передачи на ВУ значений и состояния "простых" аналоговых параметров
/// Автор: 			Chekmarev
/// Версия: 			00.00.00
/// Проект: 			КА107
{attribute 'qualified_only' := ''}
{attribute 'symbol' := 'read'}
VAR_GLOBAL	
	{attribute 'export' := '("archive":"False","communication":("cycle":"base"),"journal":"False","name":("full":"Объемная производительность","short":""),"unit":("engineering":"м3/с","electrical":""),"tag":("full":"","short":""),"digit":"1","group":"")'}
	prod     : Taspar;  // объемная производительность, м3/с
	{attribute 'export' := '("archive":"False","communication":("cycle":"base"),"journal":"False","name":("full":"Комм. производительность","short":""),"unit":("engineering":"млн·нм3/сут","electrical":""),"tag":("full":"","short":""),"digit":"1","group":"")'}
	prodCom  : Taspar; // коммерческая производительность, млн·нм3/сут
	{attribute 'export' := '("archive":"False","communication":("cycle":"base"),"journal":"False","name":("full":"Комм. производительность","short":""),"unit":("engineering":"нм3/ч","electrical":""),"tag":("full":"","short":""),"digit":"1","group":"")'}
  	Qc       : Taspar; // коммерческая производительность, нм3/ч
	{attribute 'export' := '("archive":"False","communication":("cycle":"base"),"journal":"False","name":("full":"Степень сжатия","short":""),"unit":("engineering":"","electrical":""),"tag":("full":"","short":""),"digit":"1","group":"")'}
  	pressRatio: Taspar;
	{attribute 'export' := '("archive":"False","communication":("cycle":"base"),"journal":"False","name":("full":"Нормированная частота вращения Н","short":""),"unit":("engineering":"","electrical":""),"tag":("full":"","short":""),"digit":"1","group":"АПР")'}
  	NstNorm  : Taspar;
	{attribute 'export' := '("archive":"True","communication":("cycle":"base"),"journal":"False","name":("full":"Помпажный запас","short":""),"unit":("engineering":"%","electrical":""),"tag":("full":"","short":""),"digit":"1","group":"АПР")'}
  	surgeRes : Taspar;
	{attribute 'export' := '("archive":"False","communication":("cycle":"base"),"journal":"False","name":("full":"Скорость изменения перепада на конфузоре","short":""),"unit":("engineering":"","electrical":""),"tag":("full":"","short":""),"digit":"1","group":"АПР")'}
  	ddPconf  : Taspar; // производная перепада давления на конфузоре нагнетателя по времени
	{attribute 'export' := '("archive":"False","communication":("cycle":"base"),"journal":"False","name":("full":"Скорость изменения Н","short":""),"unit":("engineering":"","electrical":""),"tag":("full":"","short":""),"digit":"1","group":"АПР")'}
  	dNst	 : Taspar;
END_VAR
(* global variable list bn *)
{attribute 'qualified_only' := ''}
{attribute 'symbol' := 'none'}
VAR_GLOBAL
	delay_filling	: REAL;
	VVN_OFF			: TON := ( PT := TIME#5M );
	ENBN			: Tsetpoint1 := ( hyst := 5, isH := 0 );
	ENBN_HR			: Tsetpoint1 := ( setpoint_value := 6, hyst := 5, isH := 0 );
	/// Кнопка стабилизации СТ
	{attribute 'symbol' := 'readwrite'}
	stabSTbtn: BOOL := TRUE;
END_VAR
(* global variable list plc *)
{attribute 'qualified_only' := ''}
VAR_GLOBAL
	BEO: Tpulse;
END_VAR
(* global variable list engine *)
{attribute 'qualified_only' := ''}
{attribute 'symbol' := 'none'}
VAR_GLOBAL
	AZ_off	: TOF := (PT := TIME#10S0MS);
	VNAheat	: Tsetpoint1 := ( setpoint_value := 5, hyst := 3, isH := 0 );
	ENBDN	: Tsetpoint1 := ( hyst := 5, isH := 0);
	ENBDN_HR: Tsetpoint1 := ( setpoint_value := 6, hyst := 5, isH := 0 );
	
	KPV1du	: TEdgeDetect;
	KPV1on	: TEdgeDetect;
	KPV1off	: TEdgeDetect;
	KPV2du	: TEdgeDetect;
	KPV2on	: TEdgeDetect;
	KPV2off	: TEdgeDetect;
	KPV3du	: TEdgeDetect;
	KPV3on	: TEdgeDetect;
	KPV3off	: TEdgeDetect;
	KPV5du	: TEdgeDetect;
	KPV5on	: TEdgeDetect;
	KPV5off	: TEdgeDetect;
	
